Omron CX-Programmer project NewProject (CX-Programmer 9.61)

# PLC NewPLC1: CP1L M

## Global symbols (name address type ; comment)
49.00 BOOL  ; Memória para fazer um movimento horizontal P2 em velocidade lenta até box.
C0017 BOOL  ; Reconhece peça On PH9: st_su_traino_bancalino_deposito_pinza_1.
C0018 BOOL  ; Reconhece peça Off PH9: st_su_traino_bancalino_deposito_pinza_1.
C0350 BOOL  ; Contagem planos mesa de rolos Pinça 2.
H0.06 BOOL  ; Bloqueio descida da ventosa sobre pilha na rulliera (Para formato 120 x 120).
H15.00 BOOL  ; Habilitação formato 120x120 Pinça 1.
T0017 BOOL  ; Reconhece peça On PH9: st_su_traino_bancalino_deposito_pinza_1.
T0018 BOOL  ; Reconhece peça Off PH9: st_su_traino_bancalino_deposito_pinza_1.
T0019 BOOL  ; Tempo desabilita HR0.06 (Habilitação formato 120 x 120).
T0682 BOOL  ; Auxiliar em função da retirada da ftc. PH3: st_pinza_1_ftc_fermata_polmone_3.
T0683 BOOL  ; Auxiliar sobe lento centro.
W0.11 BOOL  ; Reconhece peça sob PH9: st_su_traino_bancalino_deposito_pinza_1.
BIT_11200 112.00 BOOL  ; U32: pinza 1 discesa.
BIT_11201 112.01 BOOL  ; U32: pinza 1 veloce sollevamento.
BIT_11202 112.02 BOOL  ; U41: pinza 2 traslazione_lato_dx / KM9: disponibile.
BIT_11203 112.03 BOOL  ; U41: pinza 2 traslazione_lato_sx / KATB: bareira segurança.
BIT_11204 112.04 BOOL  ; U42: pinza 2 salita.
BIT_11205 112.05 BOOL  ; U42: pinza 2 discesa.
BIT_11207 112.07 BOOL  ; KM32F: pinza 1 freno sollevamento.
BIT_4500 45.00 BOOL  ; Memória Entrada Habilitada Ret Lento SX
BIT_4600 46.00 BOOL  ; Memória Entrada Habilitada Ret Lento DX
BIT_4700 47.00 BOOL  ; Lento Ventosa 1
BIT_4800 48.00 BOOL  ; Exclusão por falta peça SX
BIT_4801 48.01 BOOL  ; Exclusão por falta peça DX
BIT_900 9.00 BOOL  ; SA1: st_ripristino
BIT_901 9.01 BOOL  ; SA2: st_selettore_manuale
BIT_902 9.02 BOOL  ; PM: st_pulsante_marcia
BIT_903 9.03 BOOL  ; PA: st_pulsante_arresto
BIT_904 9.04 BOOL  ; PRA: st_pulsante_reset
BIT_905 9.05 BOOL  ; PX20: st_pinza_1_finecorsa_lato_carico
BIT_906 9.06 BOOL  ; PX21: st_pinza_1_finecorsa_lato_scaric
BIT_907 9.07 BOOL  ; PX22: st_pinza_1_finecorsa_alto
BIT_908 9.08 BOOL  ; PX2: st_pinza_1_finecorsa_basso
BIT_909 9.09 BOOL  ; PH100: st_pinza_1_ftc_per_troppo_pieno_trasporti_uscita
BIT_910 9.10 BOOL  ; PB: st_pinza_1_pulsante_comando_ribaltino
BIT_911 9.11 BOOL  ; CS_Valle: st_consenso_da_valle
CH_A270_Canal_A A270 CHANNEL  ; quota_asse_verticale_pinza2
CH_A271_Canal_B A271 CHANNEL  ; quota_asse_verticale_pinza2
CH_A272_Canal_A A272 CHANNEL  ; quota_asse_verticale_pinza1
CH_A273_Canal_B A273 CHANNEL  ; quota_asse_verticale_pinza1
CNT_100 C0100 BOOL  ; ritardo_fermata_pila_pinza1
CNT_102 C0102 BOOL  ; ritardo_per_deposito_dopo_lettura_ftc_pinza1
CNT_112 C0112 BOOL  ; conteggio_per_deposito_dopo_lettura_ftc_pinza2
CNT_20 C0020 BOOL  ; conteggio_per_stacco_pile
CNT_200 C0200 BOOL  ; intasamento_trasporto_uscita
DM_0 D0 CHANNEL  ; memoria_abilitazione_pinza1
DM_1 D1 CHANNEL  ; memoria_abilitazione_pinza2
DM_10 D10 CHANNEL  ; quota_asse_verticale_pinza1
DM_100 D100 CHANNEL  ; quota_hmi_orizzontale_prelievo_pinza1
DM_102 D102 CHANNEL  ; quota_hmi_verticale_rulliera_prelievo_pinza1
DM_104 D104 CHANNEL  ; quota_hmi_orizzontale_cinghie_deposito_pinza1
DM_106 D106 CHANNEL  ; quota_hmi_verticale_cinghie _deposito_pinza1
DM_108 D108 CHANNEL  ; quot_orizzontale_prelievo_pinza1
DM_110 D110 CHANNEL  ; quota_verticale_rulliera_prelievo_pinza1
DM_112 D112 CHANNEL  ; quota_orizzontale_cinghie_deposito_pinza1
DM_114 D114 CHANNEL  ; quota_verticale_cinghie _deposito_pinza1
DM_116 D116 CHANNEL  ; offset_per_asse_orizzontale_pinza1
DM_118 D118 CHANNEL  ; offset_per_asse_verticale_pinza1
DM_12 D12 CHANNEL  ; quota_asse_orizzontale_pinza1
DM_14 D14 CHANNEL  ; quota_asse_verticale_pinza2
DM_150 D150 CHANNEL  ; tempo_aspiraz_in_prelievo_pinza1
DM_151 D151 CHANNEL  ; Tempo desc Vent 1 M10
DM_152 D152 CHANNEL  ; ritardo_fermata_pila_pinza1
DM_153 D153 CHANNEL  ; ritardo_per_deposito_dopo_lettura_ftc_pinza1
DM_154 D154 CHANNEL  ; conteggio_per_stacco_pile
DM_155 D155 CHANNEL  ; intasamento_trasporto_uscita
DM_16 D16 CHANNEL  ; quota_asse_orizzontale_pinza2
DM_160 D160 CHANNEL  ; tempo_aspiraz_in_prelievo_pinza2
DM_161 D161 CHANNEL  ; tempo_soffio_in_deposito_pinza2
DM_163 D163 CHANNEL  ; ritardo_deposito_su_attesa_pinza2
DM_165 D165 CHANNEL  ; Retardo Lento M10.
DM_2 D2 CHANNEL  ; formato_polmoni
DM_20 D20 CHANNEL  ; offset-_vert_posiz_attesa_su_prelievo_pinza1
DM_200 D200 CHANNEL  ; quota_hmi_orizzontale_prelievo_sx_pinza2
DM_202 D202 CHANNEL  ; quota_hmi_orizzontale_prelievo_dx_pinza2
DM_204 D204 CHANNEL  ; quota_hmi_orizzontale_deposito_pinza2
DM_206 D206 CHANNEL  ; quota_hmi_verticale _deposito_pinza2
DM_208 D208 CHANNEL  ; quota_hmi_verticale_fine_pallet_sx_pinza2
DM_210 D210 CHANNEL  ; quota_hmi_verticale_fine_pallet_dx_pinza2
DM_212 D212 CHANNEL  ; quota_hmi_verticale_pila_completa_pinza2
DM_214 D214 CHANNEL  ; memoria_ultimo_prelievo_pinza2
DM_216 D216 CHANNEL  ; quota_verticale_salita_dopo_prelievo_pinza2
DM_218 D218 CHANNEL  ; quota_verticale_salita_dopo_deposito_pinza2
DM_22 D22 CHANNEL  ; offset+_vert_posiz_attesa_su_prelievo_pinza1
DM_220 D220 CHANNEL  ; quota_orizzontale_prelievo_sx_pinza2
DM_222 D222 CHANNEL  ; quota_orizzontale_prelievo_dx_pinza2
DM_224 D224 CHANNEL  ; quota_orizzontale_deposito_pinza2
DM_226 D226 CHANNEL  ; quota_verticale _deposito_pinza2
DM_228 D228 CHANNEL  ; quota_verticale_fine_pallet_sx_pinza2
DM_230 D230 CHANNEL  ; quota_verticale_fine_pallet_dx_pinza2
DM_232 D232 CHANNEL  ; quota_verticale_pila_completa_pinza2
DM_234 D234 CHANNEL  ; offset_per_asse_orizzontale_pinza2
DM_236 D236 CHANNEL  ; offset_per_asse_verticale_pinza2
DM_24 D24 CHANNEL  ; offset-_orizz_posiz_attesa_su_prelievo_pinza1
DM_250 D250 CHANNEL  ; offset-_orizz_posiz_attesa_su_deposito_pinza2
DM_252 D252 CHANNEL  ; offset+_orizz_posiz_attesa_su_deposito_pinza2
DM_254 D254 CHANNEL  ; offset-_vert_posiz_attesa_su_deposito_pinza2
DM_256 D256 CHANNEL  ; offset+_vert_posiz_attesa_su_deposito_pinza2
DM_258 D258 CHANNEL  ; offset-_orizz_posiz_prelievo_sx_pinza2
DM_26 D26 CHANNEL  ; offset+_orizz_posiz_attesa_su_prelievo_pinza1
DM_260 D260 CHANNEL  ; offset+_orizz_posiz_prelievo_sx_pinza2
DM_262 D262 CHANNEL  ; offset-_orizz_posiz_prelievo_dx_pinza2
DM_264 D264 CHANNEL  ; offset+_orizz_posiz_prelievo_dx_pinza2
DM_266 D266 CHANNEL  ; offset-_vert_posiz_prelievo_pinza2
DM_268 D268 CHANNEL  ; offset+_vert_posiz_prelievo_pinza2
DM_270 D270 CHANNEL  ; offset-_vert_posiz_salita_dopo_prelievo_pinza2
DM_272 D272 CHANNEL  ; offset+_vert_posiz_salita_dopo_prelievo_pinza2
DM_274 D274 CHANNEL  ; offset-_orizz_posiz_deposito_pinza2
DM_276 D276 CHANNEL  ; offset+_orizz_posiz_deposito_pinza2
DM_278 D278 CHANNEL  ; offset-_vert_posiz_attesa_su_deposito_pinza2
DM_28 D28 CHANNEL  ; offset-_orizz_posiz_prelievo_pinza1
DM_280 D280 CHANNEL  ; offset+_vert_posiz_attesa_su_deposito_pinza2
DM_282 D282 CHANNEL  ; offset-_vert_posiz_deposito_pinza2
DM_284 D284 CHANNEL  ; offset+_vert_posiz_deposito_pinza2
DM_286 D286 CHANNEL  ; offset-_vert_posiz_salita_dopo_deposito_pinza2
DM_288 D288 CHANNEL  ; offset+_vert_posiz_salita_dopo_deposito_pinza2
DM_290 D290 CHANNEL  ; step_salita_pinza2
DM_30 D30 CHANNEL  ; offset+_orizz_posiz_prelievo_pinza1
DM_32 D32 CHANNEL  ; offset-_vert_posiz_prelievo_pinza1
DM_34 D34 CHANNEL  ; offset+_vert_posiz_prelievo_pinza1
DM_36 D36 CHANNEL  ; offset-_vert_posiz_salita_dopo_prelievo_pinza1
DM_38 D38 CHANNEL  ; offset
DM_40 D40 CHANNEL  ; offset-_orizz_posiz_deposito_pinza1
DM_400 D400 CHANNEL  ; hz_sollevamento_pinza1_hmi
DM_401 D401 CHANNEL  ; hz_traslazione_pinza1_hmi
DM_402 D402 CHANNEL  ; hz_sollevamento_pinza2_hmi
DM_403 D403 CHANNEL  ; hz_traslazione_pinza2_hmi
DM_42 D42 CHANNEL  ; offset+_orizz_posiz_deposito_pinza1
DM_44 D44 CHANNEL  ; offset-_vert_posiz_attesa_su_deposito_pinza1
DM_450 D450 CHANNEL  ; hz_sollevamento_pinza1_fb
DM_451 D451 CHANNEL  ; hz_traslazione_pinza1_fb
DM_452 D452 CHANNEL  ; hz_sollevamento_pinza2_fb
DM_453 D453 CHANNEL  ; hz_traslazione_pinza2_fb
DM_46 D46 CHANNEL  ; offset+_vert_posiz_attesa_su_deposito_pinza1
DM_48 D48 CHANNEL  ; offset-_vert_posiz_deposito_pinza1
DM_50 D50 CHANNEL  ; offset+_vert_posiz_deposito_pinza1
DM_52 D52 CHANNEL  ; offset-_vert_posiz_salita_dopo_deposito_pinza1
DM_54 D54 CHANNEL  ; offset+_vert_posiz_salita_dopo_deposito_pinza1
DM_56 D56 CHANNEL  ; memoria_ultimo_prelievo_pinza1
DM_58 D58 CHANNEL  ; quota_verticale_salita_dopo_prelievo_pinza1
DM_60 D60 CHANNEL  ; quota_verticale_salita_dopo_deposito_pinza1
DM_62 D62 CHANNEL  ; step_salita_pinza1
HR_0 H0.00 BOOL  ; all_scatto_termico
HR_1 H0.01 BOOL  ; all_inverter
HR_10 H0.10 BOOL  ; Allarme schiacciamento pinza 2.
HR_100 H1.00 BOOL  ; azzerare_assi_pinza2
HR_1000 H10.00 BOOL  ; memoria_conteggio_avvenuto
HR_105 H1.05 BOOL  ; all_pallet_sx_finito
HR_106 H1.06 BOOL  ; all_pallet_dx_finito
HR_107 H1.07 BOOL  ; all_mancanza_pallet
HR_108 H1.08 BOOL  ; all_intrusione_area_sx
HR_109 H1.09 BOOL  ; all_intrusione_area_dx
HR_11 H0.11 BOOL  ; all_intasamento_trasporto_uscita
HR_110 H1.10 BOOL  ; all_micro_sicurezza.
HR_111 H1.11 BOOL  ; all_micro_tasteggio pinza 2.
HR_2 H0.02 BOOL  ; all_aria_compressa
HR_212 H2.12 BOOL  ; Trida_Controle lento nas 3 posições_Sempre On_020323.
HR_213 H2.13 BOOL  ; Trida_Sempre Off_010323.
HR_214 H2.14 BOOL  ; Trida_Sempre Off_050522.
HR_215 H2.15 BOOL  ; Trida_Altura ventosa_210519 (Sempre On).
HR_3 H0.03 BOOL  ; all_consenso_da_valle
HR_4 H0.04 BOOL  ; all_emergenza
HR_5 H0.05 BOOL  ; azzerare_assi_pinza1
HR_50103 H501.03 BOOL  ; polmone_completo
HR_50104 H501.04 BOOL  ; spostamento_quadrotta_da_polmone_a_prelievo
HR_50105 H501.05 BOOL  ; filtro_su_ftc_per_reset_traslazione_quadrotta
HR_8 H0.08 BOOL  ; Allarme micro tasteggio pinza 2.
HR_9 H0.09 BOOL  ; Allarme sicurezza traslazione pinza 2.
IN_0 0.00 BOOL  ; BQ1: Canale A (CH-A270) encoder sollevamento pinza 1.
IN_1 0.01 BOOL  ; BQ1: Canale B (CH-A270) encoder sollevamento pinza 1.
IN_10 0.10 BOOL  ; KABDX: st_pinza_2_barriera_dx_ripristinata (Centralina KABDX - Ok!).
IN_100 1.00 BOOL  ; SQDX: st_pinza_2_sensore_muting_dx (Fc. On durante deslocamento P2 para direita).
IN_101 1.01 BOOL  ; Allarme inverter.
IN_102 1.02 BOOL  ; $?St$Bk?_#[4] / PX102: Ft. Sobreposta Polmone 7 (Ftc. "aérea").$?St$Bk?_#[4]
IN_103 1.03 BOOL  ; Ch. habilitação formato 120 x 120.
IN_104 1.04 BOOL  ; PX104: Intasamento M11 (KM11: traino bancalino deposito pinza 1.) (Parece desativada).
IN_105 1.05 BOOL  ; CH106: parada parcial P1.
IN_106 1.06 BOOL  ; CH106: parada parcial P2.
IN_107 1.07 BOOL  ; Disponibili.
IN_108 1.08 BOOL  ; PE: Bt. emergência.
IN_109 1.09 BOOL  ; Disponibili.
IN_11 0.11 BOOL  ; SQSX: st_pinza_2_sensore_muting_sx (Fc. On durante deslocamento P2 para esquerda).
IN_110 1.10 BOOL  ; SQ100: st_pinza_1_tasteggio_1_presenza_piastrella
IN_111 1.11 BOOL  ; SQ101: st_pinza_1_tasteggio_2_finecorsa.
IN_2 0.02 BOOL  ; BQ2: Canale A (CHA-272) encoder sollevamento pinza 2.
IN_200 2.00 BOOL  ; Disponibili.
IN_201 2.01 BOOL  ; PH1: st_pinza_1_ftc_fermata_polmone_1: bancal operatore (Ribaltatore) (Não tem).
IN_202 2.02 BOOL  ; PH2: st_pinza_1_ftc_fermata_polmone_2.
IN_203 2.03 BOOL  ; PH3: st_pinza_1_ftc_fermata_polmone_3 (Não tem).
IN_204 2.04 BOOL  ; PH4: st_pinza_1_ftc_fermata_polmone_4.
IN_205 2.05 BOOL  ; PH5: st_pinza_1_ftc_fermata_polmone_5.
IN_206 2.06 BOOL  ; PH6: st_pinza_1_ftc_fermata_polmone_6 (Não tem).
IN_207 2.07 BOOL  ; PH7: st_pinza_1_ftc_fermata_polmone_7_lettura_lunghezza_pila (Não tem).
IN_208 2.08 BOOL  ; PH8: st_pinza_1_ftc_fermata_polmone_8_prelievo_pinza_1.
IN_209 2.09 BOOL  ; PH9: st_su_traino_bancalino_deposito_pinza_1.
IN_210 2.10 BOOL  ; PX30: st_reed_ribaltino_alto.
IN_211 2.11 BOOL  ; PX31: st_reed_ribaltino_basso.
IN_3 0.03 BOOL  ; BQ2: Canale B (CHA-272) encoder sollevamento pinza 2.
IN_300 3.00 BOOL  ; P1/P2: st_pressostati.
IN_301 3.01 BOOL  ; PX32: st_pinza_2_finecorsa_lato_pedana_sx.
IN_302 3.02 BOOL  ; PX33: st_pinza_2_finecorsa_lato_pedana_dx.
IN_303 3.03 BOOL  ; PX34: st_pinza_2_finecorsa_alto.
IN_304 3.04 BOOL  ; PX35: st_pinza_2_finecorsa_basso.
IN_305 3.05 BOOL  ; PX36: st_pinza_2_tasteggio_1_presenza_piastrella.
IN_306 3.06 BOOL  ; PH10: st_pinza_2_ftc_presenza_pallet_sx (Sempre On).
IN_307 3.07 BOOL  ; PH11: st_pinza_2_ftc_presenza_pallet_dx (Sempre On).
IN_308 3.08 BOOL  ; P8: st_pinza_2_pulsante_richiesta_accesso_Pedana_sx.
IN_309 3.09 BOOL  ; P9: st_pinza_2_pulsante_richiesta_accesso_pedana_dx.
IN_310 3.10 BOOL  ; Px37: st_pinza_2_tasteggio_2_finecorsa.
IN_311 3.11 BOOL  ; Disponibili.
IN_4 0.04 BOOL  ; BQ3: Canale A (DM14) encoder traslazione pinza 1.
IN_400 4.00 BOOL  ; SA3: st_pinza 2_selettore_esclusione pallet sx.
IN_401 4.01 BOOL  ; SA4: st_pinza 2_selettore_esclusione pallet dx.
IN_402 4.02 BOOL  ; PF: st_pinza 2_pulsante_pila finita.
IN_403 4.03 BOOL  ; PX13: st_pinza_2_presenza_piastrelle.
IN_404 4.04 BOOL  ; Disponibili.
IN_405 4.05 BOOL  ; Disponibili.
IN_406 4.06 BOOL  ; Disponibili.
IN_407 4.07 BOOL  ; Disponibili.
IN_408 4.08 BOOL  ; Disponibili.
IN_409 4.09 BOOL  ; Disponibili.
IN_410 4.10 BOOL  ; Disponibili.
IN_411 4.11 BOOL  ; Disponibili.
IN_5 0.05 BOOL  ; BQ3: Canale B (DM14) encoder traslazione pinza 1.
IN_500 5.00 BOOL  ; SA1: st_ripristino (Sempre On_Jump +).
IN_501 5.01 BOOL  ; SA2: selettore manuale/automatico.
IN_502 5.02 BOOL  ; PM: st_pulsante_marcia.
IN_503 5.03 BOOL  ; PA: st_pulsante_arresto.
IN_504 5.04 BOOL  ; PRA: st_pulsante_reset_allarmi.
IN_505 5.05 BOOL  ; PX20: st_pinza_1_finecorsa_lato_carico.
IN_506 5.06 BOOL  ; PX21: st_pinza_1_finecorsa_lato_scarico.
IN_507 5.07 BOOL  ; PX22: st_pinza_1_finecorsa_alto.
IN_508 5.08 BOOL  ; PX23: st_pinza_1_finecorsa_basso.
IN_509 5.09 BOOL  ; PH100: st_pinza_1_ftc_per_troppo_pieno_trasporti_uscita (Sempre Off_Nada ligado nesta entrada).
IN_510 5.10 BOOL  ; PB: st_pinza_1_pulsante_comando_ribaltino.
IN_511 5.11 BOOL  ; CS_Valle: st_consenso_da_valle.
IN_6 0.06 BOOL  ; BQ4: Canale A (DM16) encoder traslazione pinza 2.
IN_7 0.07 BOOL  ; BQ4: Canale B  (DM16) encoder traslazione pinza 2.
IN_8 0.08 BOOL  ; Allarme termico motori.
IN_9 0.09 BOOL  ; KABSX: St_pinza_2_barriera_sx_ripristinata (Centralina KABSX - Ok!).
OUT_10000 100.00 BOOL  ; KA10: consenso a monte.
OUT_10001 100.01 BOOL  ; HA1: sirena.
OUT_10002 100.02 BOOL  ; HL5: spia allarme.
OUT_10003 100.03 BOOL  ; U32: pinza 1 discesa.
OUT_10004 100.04 BOOL  ; U32: pinza 1 veloce sollevamento.
OUT_10005 100.05 BOOL  ; HL8: spia acesso consentito sx.
OUT_10006 100.06 BOOL  ; HL9: spia acesso consentito dx.
OUT_10007 100.07 BOOL  ; HL10: spia segnalazione pedana sx finita.
OUT_10100 101.00 BOOL  ; HL11: spia segnalazione pedana dx finita.
OUT_10101 101.01 BOOL  ; KM21: pompa vuoto pinza 1.
OUT_10102 101.02 BOOL  ; KA22: pompa vuoto pinza 2.
OUT_10103 101.03 BOOL  ; Clock peças produzidas (Sobre painel Spaccatrice).
OUT_10104 101.04 BOOL  ; U31: pinza 1 traslazione lato scarico.
OUT_10105 101.05 BOOL  ; U31: pinza 1 traslazione lato carico.
OUT_10106 101.06 BOOL  ; U31: pinza 1 veloce traslazione.
OUT_10107 101.07 BOOL  ; U32: pinza1 salita.
OUT_10199 102.00 BOOL  ; Reserva (Desenho elétrico: KM41F: freno traslazione pinza 2).
OUT_10200 102.01 BOOL  ; KM42F: pinza 2 freno solevamento.
OUT_10201 102.02 BOOL  ; KM1: polmone 1: bancalino operatore (Ribaltatore).
OUT_10202 102.03 BOOL  ; KM2: polmone 2.
OUT_10203 102.04 BOOL  ; KM3: polmone 3.
OUT_10204 102.05 BOOL  ; KM4: polmone 4.
OUT_10205 102.06 BOOL  ; KM5: polmone 5.
OUT_10206 102.07 BOOL  ; KM6: polmone 6.
OUT_10300 103.00 BOOL  ; KM7: polmone 7.
OUT_10301 103.01 BOOL  ; KM8: polmone 8 (Sotto pinza 1).
OUT_10302 103.02 BOOL  ; U41: pinza 2 traslazione_lato_dx / KM9: disponibile.
OUT_10303 103.03 BOOL  ; KM10 / KA10403: disponíbile.
OUT_10304 103.04 BOOL  ; KM11: traino bancalino deposito pinza 1.
OUT_10305 103.05 BOOL  ; KM15: disponibile.
OUT_10306 103.06 BOOL  ; U41: pinza 2 traslazione_lato_sx / KATB: barreira segurança.
OUT_10307 103.07 BOOL  ; KASX: acesso pedana sx (On: liberado acesso).
OUT_10400 104.00 BOOL  ; KADX: acesso pedana dx (On: liberado acesso).
OUT_10401 104.01 BOOL  ; KAYV1: ev. salita bancalino operatore.
OUT_10402 104.02 BOOL  ; KAYV2: ev. discesa bancalino operatore.
OUT_10403 104.03 BOOL  ; KAYV3: ev. aspirazione pinza 1.
OUT_10404 104.04 BOOL  ; KAYV4: ev. soffio pinza 1.
OUT_10405 104.05 BOOL  ; KAYV5: ev. aspirazione pinza 2.
OUT_10406 104.06 BOOL  ; KAYV6: ev. soffio pinza 2.
OUT_10407 104.07 BOOL  ; KA10505: disponibile.
OUT_10500 105.00 BOOL  ; Disponibile.
OUT_10501 105.01 BOOL  ; HL12: spia marcia.
OUT_10502 105.02 BOOL  ; U41: pinza 2 veloce traslazione.
OUT_10503 105.03 BOOL  ; U42: pinza 2 veloce solevamento.
OUT_10504 105.04 BOOL  ; U42: pinza 2 salita.
OUT_10505 105.05 BOOL  ; U42: pinza 2 discesa.
OUT_10506 105.06 BOOL  ; Disponibile.
OUT_10507 105.07 BOOL  ; KM32F: pinza 1 freno sollevamento.
TIM_100 T0100 BOOL  ; tempo_aspiraz_in_prelievo_pinza1
TIM_101 T0101 BOOL  ; tempo_soffio_in_deposito_pinza1 Antigo D151
TIM_103 T0103 BOOL  ; attesa_per_rideposito_pinza1
TIM_110 T0110 BOOL  ; tempo_aspiraz_in_prelievo_pinza2
TIM_111 T0111 BOOL  ; tempo_soffio_in_deposito_pinza2
TIM_123 T0123 BOOL  ; attesa_per_rideposito_pinza2
TIM_15 T0015 BOOL  ; Retardo conta peça produzida.
TIM_16 T0016 BOOL  ; Tempo permanência pulso clock.
TIM_20 T0020 BOOL  ; standby_aspiratore_pinza1
TIM_21 T0021 BOOL  ; standby_aspiratpore_pinza2
TIM_25 T0025 BOOL  ; Ret Stop tração de saida
TIM_26 T0026 BOOL  ; Ret FTC Px102 Separa Fila
TIM_27 T0027 BOOL  ; Retardo Lento M10.
TIM_29 T0029 BOOL  ; Tempo Para desligar Bombas com Emergencia
TIM_3 T0003 BOOL  ; Ritardo off st_pinza_1_ftc_fermata_polmone_8_prelievo_pinza_1.
TIM_30 T0030 BOOL  ; Retardo Mivimento Palet Dx Painel
TIM_31 T0031 BOOL  ; Retardo conta peça produzida.
TIM_32 T0032 BOOL  ; Ret. Libera Movimento Palet SX
TIM_33 T0033 BOOL  ; Ret Libera Movimento Palet DX
TIM_34 T0034 BOOL  ; Fim Pilha manual
TIM_35 T0035 BOOL  ; Plano vazio Ventosa 2
TIM_36 T0036 BOOL  ; Ret Leitura Hor SX
TIM_37 T0037 BOOL  ; Ret Leitura Hor DX
TIM_38 T0038 BOOL  ; Retardo libera parada parcial P1.
TIM_39 T0039 BOOL  ; Retardo libera parada parcial P2.
TIM_4 T0004 BOOL  ; Ritardo st_consenso_da_valle
TIM_5 T0005 BOOL  ; Ritardo riconosce pila finita manuale.
TIM_6 T0006 BOOL  ; Ritardo uscita di automatico.
TIM_650 T0650 BOOL  ; ritardo_rich_acc_sx
TIM_651 T0651 BOOL  ; ritardo_rich_acc_dx
TIM_652 T0652 BOOL  ; Ret Libera Acesso DX
TIM_653 T0653 BOOL  ; Ret Libera Acesso SX
TIM_7 T0007 BOOL  ; Ritardo riconosce ftc fermata polmone 6_7.
TIM_8 T0008 BOOL  ; Allarme micro tasteggio pinza 2.
W_0 W0.00 BOOL  ; st_ripristino
W_1 W0.01 BOOL  ; st_scatto_termico
W_10 W0.10 BOOL  ; st_consenso_da_valle senza tempo
W_100 W1.00 BOOL  ; st_pinza_1_finecorsa_lato_carico
W_1000 W10.00 BOOL  ; spia_marcia
W_10000 W100.00 BOOL  ; attesa_per_accesso_sx
W_10002 W100.02 BOOL  ; posizionamento_al_centro_da_rich_acc_sx_dx
W_10003 W100.03 BOOL  ; attesa_sx_con_pinza_a_dx
W_10004 W100.04 BOOL  ; accesso_consentito_a_sx
W_10006 W100.06 BOOL  ; attesa_sx_con_pinza_a_sx
W_1001 W10.01 BOOL  ; spia_allarme
W_10013 W100.13 BOOL  ; allarme_fermo_ciclo
W_10014 W100.14 BOOL  ; tacita_sirena
W_1002 W10.02 BOOL  ; sirena
W_1003 W10.03 BOOL  ; consenso_a_monte
W_101 W1.01 BOOL  ; st_pinza_1_finecorsa_lato_scarico
W_10100 W101.00 BOOL  ; attesa_per_accesso_dx
W_10102 W101.02 BOOL  ; ok_accesso
W_10103 W101.03 BOOL  ; attesa_dx_con_pinza_a_sx
W_10104 W101.04 BOOL  ; accesso_consentito_a_dx
W_10106 W101.06 BOOL  ; attesa_dx_con_pinza_a_dx
W_102 W1.02 BOOL  ; st_pinza_1_rallentamento_lato_carico
W_10203 W102.03 BOOL  ; attesa_ripresa_ciclo
W_103 W1.03 BOOL  ; st_pinza_1_rallentamento_lato_scarico
W_104 W1.04 BOOL  ; st_pinza_1_finecorsa_alto
W_105 W1.05 BOOL  ; st_pinza_1_finecorsa_basso
W_106 W1.06 BOOL  ; st_pinza_1_tasteggio_1_presenza_piastrella
W_107 W1.07 BOOL  ; st_pinza_1_tasteggio_2_finecorsa
W_108 W1.08 BOOL  ; st_pinza_1_ftc_fermata_polmone_8_prelievo_pinza_1.
W_109 W1.09 BOOL  ; st_pinza_1_ftc_lettura_lunghezza_pila
W_110 W1.10 BOOL  ; $?St$Bk?_#[5] / PX102: Ft. Sobreposta Polmone 7 (Ftc. "aérea").$?St$Bk?_#[5]
W_1100 W11.00 BOOL  ; pinza_1_traslazione_verso_carico
W_11000 W110.00 BOOL  ; vel_rallentata_sollevamento_pinza1
W_11001 W110.01 BOOL  ; vel_rallentata_traslazione_pinza1
W_11002 W110.02 BOOL  ; finecorsa_lato_prelievo_pinza1
W_11003 W110.03 BOOL  ; finecorsa_lato_deposito_pinza1
W_1101 W11.01 BOOL  ; pinza_1_traslazione_verso_scarico
W_1102 W11.02 BOOL  ; pinza_1_salita
W_1103 W11.03 BOOL  ; pinza_1_discesa
W_1104 W11.04 BOOL  ; pinza_1_ev_aspirazione
W_1105 W11.05 BOOL  ; pinza_1_ev_soffio
W_1106 W11.06 BOOL  ; pinza_1_aspiratore
W_1107 W11.07 BOOL  ; pinza_1_trasporto1_cinghie
W_1108 W11.08 BOOL  ; pinza_1_trasporto2_cinghie
W_1109 W11.09 BOOL  ; pinza_1_trasporto3_cinghie
W_111 W1.11 BOOL  ; PH5: st_pinza_1_ftc_fermata_polmone_5 (Sem função no programa).
W_1110 W11.10 BOOL  ; Polmone 8 (Sotto pinza 1)_manual.
W_1111 W11.11 BOOL  ; Polmone 7_manual.
W_1112 W11.12 BOOL  ; Polmone 6_manual.
W_1113 W11.13 BOOL  ; Polmone 5_manual.
W_1114 W11.14 BOOL  ; Polmone 4_manual.
W_1115 W11.15 BOOL  ; Polmone 3_manual.
W_112 W1.12 BOOL  ; PH4: st_pinza_1_ftc_fermata_polmone_4.
W_113 W1.13 BOOL  ; PH5: st_pinza_1_ftc_fermata_polmone_5.
W_114 W1.14 BOOL  ; PH2: st_pinza_1_ftc_fermata_polmone_2.
W_115 W1.15 BOOL  ; PH1: st_pinza_1_ftc_fermata_polmone_1: bancal operatore (Ribaltatore) (Não tem).
W_1200 W12.00 BOOL  ; Polmone 2_manual.
W_1201 W12.01 BOOL  ; pinza_1_rulliera_8
W_1202 W12.02 BOOL  ; Polmone 1: bancalino operatore (Ribaltatore)_manual.
W_1203 W12.03 BOOL  ; pinza_1_ev_salita_ribaltino
W_1204 W12.04 BOOL  ; pinza_1_ev_discesa_ribaltino
W_1300 W13.00 BOOL  ; pinza_2_traslazione_da_sx_a_dx
W_1301 W13.01 BOOL  ; pinza_2_traslazione_da_dx_a_sx
W_1302 W13.02 BOOL  ; pinza_2_salita
W_1303 W13.03 BOOL  ; pinza_2_discesa
W_1304 W13.04 BOOL  ; pinza_2_ev_aspirazione
W_1305 W13.05 BOOL  ; pinza_2_ev_soffio
W_1306 W13.06 BOOL  ; pinza_2_aspiratore
W_1307 W13.07 BOOL  ; pinza_2_trasporto1_cinghie
W_1308 W13.08 BOOL  ; pinza_2_trasporto2_cinghie
W_1309 W13.09 BOOL  ; pinza_2_trasporto3_cinghie
W_1310 W13.10 BOOL  ; pinza_2_rulliera_1_deposito
W_1311 W13.11 BOOL  ; pinza_2_rulliera_2
W_1312 W13.12 BOOL  ; pinza_2_rulliera_3
W_1313 W13.13 BOOL  ; pinza_2_trasporto_rulli_deviatore
W_1314 W13.14 BOOL  ; pinza_2_trasporto_cinghie_deviatore
W_1315 W13.15 BOOL  ; pinza_2_ev_deviatore
W_1400 W14.00 BOOL  ; pinza_2_spia_pallet_sx_finito
W_1401 W14.01 BOOL  ; pinza_2_spia_pallet_dx_finito
W_1402 W14.02 BOOL  ; pinza_2_bypass_barriera_sx
W_1403 W14.03 BOOL  ; pinza_2_bypass_barriera_dx
W_1404 W14.04 BOOL  ; pinza_2_spia_accesso_consentito_sx
W_1405 W14.05 BOOL  ; pinza_2_spia_accesso_consentito_dx
W_2 W0.02 BOOL  ; st_allarme_inverter
W_200 W2.00 BOOL  ; st_pinza_1_ftc_fermata_polmone_8
W_2000 W20.00 BOOL  ; spia_marcia_automatico
W_20000 W200.00 BOOL  ; tasto_azzera_assi_pinza1
W_2001 W20.01 BOOL  ; spia_allarme_automatico
W_2002 W20.02 BOOL  ; sirena_automatico
W_2003 W20.03 BOOL  ; consenso_a_monte_automatico
W_201 W2.01 BOOL  ; st_pinza_1_ftc_fermata_polmone_9
W_202 W2.02 BOOL  ; st_pinza_1_pulsante_comando_ribaltino
W_203 W2.03 BOOL  ; st_pinza_1_reed_ribaltino_alto
W_204 W2.04 BOOL  ; st_pinza_1_reed_ribaltino_basso
W_205 W2.05 BOOL  ; PH9: st_su_traino_bancalino_deposito_pinza_1.
W_20500 W205.00 BOOL  ; tasto_azzera_assi_pinza2
W_206 W2.06 BOOL  ; st_pinza_1_ftc_per_troppo_pieno_trasporti_uscita
W_207 W2.07 BOOL  ; st_pinza 2_pulsante_pila finita.
W_208 W2.08 BOOL  ; Sensor presença peça pinza 2.
W_2100 W21.00 BOOL  ; pinza_1_traslazione_verso_carico_automatico
W_21000 W210.00 BOOL  ; vel_rallentata_sollevamento_pinza2
W_21001 W210.01 BOOL  ; vel_rallentata_traslazione_pinza2
W_21002 W210.02 BOOL  ; vel_rallentata_traslazione_pinza2.
W_21003 W210.03 BOOL  ; vel_rallentata_traslazione_pinza2.
W_21004 W210.04 BOOL  ; vel_rallentata_traslazione_pinza2.
W_2101 W21.01 BOOL  ; pinza_1_traslazione_verso_scarico_automatico
W_2102 W21.02 BOOL  ; pinza_1_salita_automatico
W_2103 W21.03 BOOL  ; pinza_1_discesa_automatico
W_2104 W21.04 BOOL  ; pinza_1_ev_aspirazione_automatico
W_2105 W21.05 BOOL  ; pinza_1_ev_soffio_automatico
W_2106 W21.06 BOOL  ; pinza_1_aspiratore_automatico
W_2107 W21.07 BOOL  ; pinza_1_trasporto1_cinghie_automatico
W_2108 W21.08 BOOL  ; pinza_1_trasporto2_cinghie_automatico
W_2109 W21.09 BOOL  ; pinza_1_trasporto3_cinghie_automatico
W_2110 W21.10 BOOL  ; Polmone 8 (Sotto pinza 1)_automatico.
W_21109 W211.09 BOOL  ; posiizonam_al_centro_per_accesso_pinza2
W_2111 W21.11 BOOL  ; Polmone 7._automatico
W_21115 W211.15 BOOL  ; controllo_richieste_accesso
W_2112 W21.12 BOOL  ; Polmone 6_automatico.
W_2113 W21.13 BOOL  ; Polmone 5_automatico.
W_2114 W21.14 BOOL  ; Polmone 4_automatico.
W_2115 W21.15 BOOL  ; Polmone 3_automatico.
W_2200 W22.00 BOOL  ; Polmone 2_automatico.
W_2201 W22.01 BOOL  ; pinza_1_rulliera_8_automatico
W_2202 W22.02 BOOL  ; Polmone 1: bancalino operatore (Ribaltatore)_ribaltino_automatico.
W_2203 W22.03 BOOL  ; pinza_1_ev_salita_ribaltino_automatico
W_2204 W22.04 BOOL  ; pinza_1_ev_discesa_ribaltino_automatico
W_2300 W23.00 BOOL  ; pinza_2_traslazione_da_sx_a_dx_automatico
W_2301 W23.01 BOOL  ; pinza_2_traslazione_da_dx_a_sx_automatico
W_2302 W23.02 BOOL  ; pinza_2_salita_automatico
W_2303 W23.03 BOOL  ; pinza_2_discesa_automatico
W_2304 W23.04 BOOL  ; pinza_2_ev_aspirazione_automatico
W_2305 W23.05 BOOL  ; pinza_2_ev_soffio_automatico
W_2306 W23.06 BOOL  ; pinza_2_aspiratore_automatico
W_2307 W23.07 BOOL  ; pinza_2_trasporto1_cinghie_automatico
W_2308 W23.08 BOOL  ; pinza_2_trasporto2_cinghie_automatico
W_2309 W23.09 BOOL  ; pinza_2_trasporto3_cinghie_automatico
W_2310 W23.10 BOOL  ; pinza_2_rulliera_1_deposito_automatico
W_2311 W23.11 BOOL  ; pinza_2_rulliera_2_automatico
W_2312 W23.12 BOOL  ; pinza_2_rulliera_3_automatico
W_2313 W23.13 BOOL  ; pinza_2_trasporto_rulli_deviatore_automatico
W_2314 W23.14 BOOL  ; pinza_2_trasporto_cinghie_deviatore_automatico
W_2315 W23.15 BOOL  ; pinza_2_ev_deviatore_automatico
W_2400 W24.00 BOOL  ; pinza_2_spia_pallet_sx_finito_automatico
W_2401 W24.01 BOOL  ; pinza_2_spia_pallet_dx_finito_automatico
W_2402 W24.02 BOOL  ; pinza_2_bypass_barriera_sx_automatico
W_2403 W24.03 BOOL  ; pinza_2_bypass_barriera_dx_automatico
W_2404 W24.04 BOOL  ; pinza_2_spia_accesso_consentito_sx_automatico
W_2405 W24.05 BOOL  ; pinza_2_spia_accesso_consentito_dx_automatico
W_27500 W275.00 BOOL  ; flag_presenza_pallet_iniziale
W_3 W0.03 BOOL  ; st_selettore_manuale
W_300 W3.00 BOOL  ; st_pinza_2_finecorsa_lato_sx
W_301 W3.01 BOOL  ; st_pinza_2_finecorsa_lato_dx
W_302 W3.02 BOOL  ; st_pinza_2_finecorsa_alto
W_303 W3.03 BOOL  ; st_pinza_2_finecorsa_basso
W_30309 W303.09 BOOL  ; pallet_sx_esaurito
W_30310 W303.10 BOOL  ; pile_finite_su_rulliera
W_30311 W303.11 BOOL  ; pallet_dx_esaurito
W_30312 W303.12 BOOL  ; Ausiliare esclusione pallet sx.
W_30313 W303.13 BOOL  ; Ausiliare esclusione pallet dx.
W_30314 W303.14 BOOL  ; Ausiliare lento prima discesa su box sx.
W_30315 W303.15 BOOL  ; Ausiliare lento prima discesa su box dx.
W_304 W3.04 BOOL  ; st_pinza_2_tasteggio_1_presenza_piastrella
W_305 W3.05 BOOL  ; st_pinza_2_tasteggio_2_finecorsa
W_306 W3.06 BOOL  ; st_pinza_2_ftc_fermata_prelievo
W_307 W3.07 BOOL  ; st_pinza_2_barriera_sx_ripristinata
W_308 W3.08 BOOL  ; st_pinza_2_barriera_dx_ripristinata
W_309 W3.09 BOOL  ; st_pinza_2_sensore_muting_sx
W_310 W3.10 BOOL  ; st_pinza_2_sensore_muting_dx
W_311 W3.11 BOOL  ; st_pinza_2_pulsante_rich_accesso_sx
W_312 W3.12 BOOL  ; st_pinza_2_pulsante_rich_accesso_dx
W_313 W3.13 BOOL  ; Ausiliare esclusione pallet sx. (Era st_pinza_2_ftc_presenza_pallet_sx).
W_314 W3.14 BOOL  ; Ausiliare esclusione pallet dx. (st_pinza_2_ftc_presenza_pallet_dx).
W_315 W3.15 BOOL  ; st_pinza_2_ftc_su_rulliera_deposito
W_35002 W350.02 BOOL  ; attesa_per_carico_a_sx
W_35003 W350.03 BOOL  ; attesa_per_carico_a_dx
W_35500 W355.00 BOOL  ; pallet_a_a_sx_finito
W_35501 W355.01 BOOL  ; pallet_a_dx_finito
W_35502 W355.02 BOOL  ; pile_finite_stop_ciclo
W_35503 W355.03 BOOL  ; Pila finita manuale.
W_39000 W390.00 BOOL  ; ok_carica_a_sx
W_39001 W390.01 BOOL  ; ok_carica_a_dx
W_4 W0.04 BOOL  ; st_selettore_automatico
W_400 W4.00 BOOL  ; st_pinza_2_ftc_ingresso_deviatore
W_4000 W40.00 BOOL  ; pronto_manuale
W_4001 W40.01 BOOL  ; stato_manuale
W_4002 W40.02 BOOL  ; pronto_automatico
W_4003 W40.03 BOOL  ; stato_automatico
W_4004 W40.04 BOOL  ; standby_pinza1
W_4005 W40.05 BOOL  ; standby_pinza2
W_4007 W40.07 BOOL  ; Retardo Sem Ciclo
W_401 W4.01 BOOL  ; st_pinza_2_ftc_deviatore
W_402 W4.02 BOOL  ; st_pinza_2_ftc_uscita_deviatore
W_403 W4.03 BOOL  ; st_pinza 2_selettore_esclusione pallet sx (On: incluso).
W_404 W4.04 BOOL  ; st_pinza 2_selettore_esclusione pallet dx (On: incluso).
W_410 W4.10 BOOL  ; Formato_1800
W_4100 W41.00 BOOL  ; ciclo_azzeramento_assi_pinza1
W_4101 W41.01 BOOL  ; fine_azzeramento_pinza1
W_4102 W41.02 BOOL  ; flag_assi_azzerati_pinza1
W_4103 W41.03 BOOL  ; salita_per_azzeramento_pinza1
W_4104 W41.04 BOOL  ; discesa_per_azzeramento_pinza1
W_4105 W41.05 BOOL  ; uscita_da_finecorsa_alto_azzeram_pinza1
W_4106 W41.06 BOOL  ; reset_salita_per_azzeramento_pinza1
W_4107 W41.07 BOOL  ; reset_discesa_per_azzeram_pinza1
W_4108 W41.08 BOOL  ; ok_per_azzermento_asse_orizz_pinza1
W_4109 W41.09 BOOL  ; traslazione_lato_carico_per_azzeramento_pinza1
W_4110 W41.10 BOOL  ; traslazione_lato_scarico_per_azzeramento_pinza1
W_4111 W41.11 BOOL  ; reset_traslazione_lato_carico_per_azzeramento_pinza1
W_4112 W41.12 BOOL  ; uscita_da_finec_lato_carico_per_azzeramento_pinza1
W_4113 W41.13 BOOL  ; reset_traslazione_lato_scarico_per_azzeramento_pinza1
W_4300 W43.00 BOOL  ; ciclo_azzeramento_assi_pinza2
W_4301 W43.01 BOOL  ; fine_azzeramento_pinza2
W_4302 W43.02 BOOL  ; flag_assi_azzerati_pinza2
W_4303 W43.03 BOOL  ; salita_per_azzeramento_pinza2
W_4304 W43.04 BOOL  ; discesa_per_azzeramento_pinza2
W_4305 W43.05 BOOL  ; uscita_da_finecorsa_alto_azzeram_pinza2
W_4306 W43.06 BOOL  ; reset_salita_per_azzeramento_pinza2
W_4307 W43.07 BOOL  ; reset_discesa_per_azzeram_pinza2
W_4308 W43.08 BOOL  ; ok_per_azzermento_asse_orizz_pinza2
W_4309 W43.09 BOOL  ; traslazione_lato_sx_per_azzeramento_pinza2
W_4310 W43.10 BOOL  ; traslazione_lato_dx_per_azzeramento_pinza2
W_4311 W43.11 BOOL  ; reset_traslazione_lato_carico_per_azzeramento_pinza2
W_4312 W43.12 BOOL  ; uscita_da_finec_lato_carico_per_azzeramento_pinza2
W_4313 W43.13 BOOL  ; reset_traslazione_lato_scarico_per_azzeramento_pinza2
W_45000 W450.00 BOOL  ; pallet_sx_sostituito
W_45001 W450.01 BOOL  ; pallet_sx_cambiato
W_45002 W450.02 BOOL  ; pallet_dx_sostituito
W_45003 W450.03 BOOL  ; pallet_dx_cambiato
W_5 W0.05 BOOL  ; st_pulsante_marcia
W_5000 W50.00 BOOL  ; start_conteggio_fermata_pila_pinza1
W_50000 W500.00 BOOL  ; start
W_50001 W500.01 BOOL  ; wr_n1
W_50002 W500.02 BOOL  ; busy_n1
W_50003 W500.03 BOOL  ; wr_n2
W_50004 W500.04 BOOL  ; busy_n2
W_50005 W500.05 BOOL  ; wr_n3
W_50006 W500.06 BOOL  ; busy_n3
W_50007 W500.07 BOOL  ; wr_n4
W_50008 W500.08 BOOL  ; busy_n4
W_5001 W50.01 BOOL  ; fermata_polmoni_per_centraggio_
W_50011 W500.11 BOOL  ; restart_write
W_5002 W50.02 BOOL  ; polmonatura_singola
W_5003 W50.03 BOOL  ; polmonatura_doppia
W_5004 W50.04 BOOL  ; polmonatura_per_quadrotta
W_505 W5.05 BOOL  ; Espelho st_pinza_2_tasteggio_2_finecorsa
W_6 W0.06 BOOL  ; st_pulsante_arresto
W_6000 W60.00 BOOL  ; abilitazione_pinza1
W_6001 W60.01 BOOL  ; richiesta_inizio_ciclo_pinza1
W_6002 W60.02 BOOL  ; pinza1_in_ciclo
W_6003 W60.03 BOOL  ; start_ciclo_pinza1
W_6008 W60.08 BOOL  ; primo_ciclo_pinza1
W_6100 W61.00 BOOL  ; posizione_attesa_su_prelievo_pinza1
W_6101 W61.01 BOOL  ; posiz_attesa_su_prelievo_discesa_pinza1
W_6102 W61.02 BOOL  ; posiz_attesa_su_prelievo_salita_pinza1
W_6103 W61.03 BOOL  ; ok_posione_verticale_attesa_pinza1
W_6104 W61.04 BOOL  ; posiz_attesa_su_prelievo_trasl_verso_deposito_pinza1
W_6105 W61.05 BOOL  ; posiz_attesa_su_prelievo_trasl_verso_carico_pinza1
W_6106 W61.06 BOOL  ; ok_posione_orizzontale_attesa_pinza1
W_6200 W62.00 BOOL  ; posizione_prelievo_asse_orizzontale_pinza1
W_6201 W62.01 BOOL  ; posiz_prelievo_trasl_verso_deposito_pinza1
W_6202 W62.02 BOOL  ; posiz_prelievo_trasl_verso_prelievo_pinza1
W_6203 W62.03 BOOL  ; ok_posione_orizzontale_prelievo_pinza1
W_6300 W63.00 BOOL  ; discesa_per_prelievo_piastrella_pinza1
W_6301 W63.01 BOOL  ; piastrella_su_ventose_pinza1
W_6302 W63.02 BOOL  ; posizione_verticale_discesa_prelievo_pinza1
W_6303 W63.03 BOOL  ; ok_posizione_verticale_prelievo_pinza1
W_6304 W63.04 BOOL  ; ok_posizione_verticale_rideposito_su_prelievo_pinza1
W_6400 W64.00 BOOL  ; prelievo_piastrella_pinza1
W_6401 W64.01 BOOL  ; aspirazione_per_prelievo_pinza1
W_6402 W64.02 BOOL  ; ok_prelievo_pinza1
W_6500 W65.00 BOOL  ; salita_dopo_prelievo_piastrella_pinza1
W_6501 W65.01 BOOL  ; posizionamento_verticale_salita_dopo_prelievo_pinza1
W_6502 W65.02 BOOL  ; posizionamento_verticale_discesa_dopo_prelievo_pinza1
W_6503 W65.03 BOOL  ; ok_posizione_verticale_dopo_prelievo_pinza1
W_6600 W66.00 BOOL  ; posizione_deposito_asse_orizzontale_pinza1
W_6601 W66.01 BOOL  ; posizionamento_orizzontale_verso_deposito_per_deposito_pinza1
W_6602 W66.02 BOOL  ; posizionamento_orizzontale_verso_prelievo_per_deposito_pinza1
W_6603 W66.03 BOOL  ; ok_posizione_orizzontale_deposito_pinza1
W_6700 W67.00 BOOL  ; discesa_per_attesa_deposito_pinza1
W_6701 W67.01 BOOL  ; posizionamento_verticale_salita_per_attesa_su_deposito_pinza1
W_6702 W67.02 BOOL  ; posizionamento_verticale_discesa_per_attesa_su_deposito_pinza1
W_6703 W67.03 BOOL  ; ok_posizionamento_verticale_attesa_deposito_pinza1
W_6800 W68.00 BOOL  ; discesa_per_deposito_piastrella_pinza1
W_6801 W68.01 BOOL  ; posizionamento_verticale_salita_per_deposito_pinza1
W_6802 W68.02 BOOL  ; posizionamento_verticale_discesa_per_deposito_pinza1
W_6803 W68.03 BOOL  ; ok_posizione_verticale_deposito_pinza1
W_6900 W69.00 BOOL  ; deposito_piastrella_pinza1
W_6901 W69.01 BOOL  ; soffio_per_deposito_pinza1
W_6902 W69.02 BOOL  ; ok_deposito_pinza1
W_7 W0.07 BOOL  ; st_pulsante_reset
W_7000 W70.00 BOOL  ; salita_dopo_deposito_pinza1
W_7001 W70.01 BOOL  ; posizionamento_verticale_salita_dopo_deposito_pinza1
W_7002 W70.02 BOOL  ; posizionamento_verticale_discesa_dopo_deposito_pinza1
W_7003 W70.03 BOOL  ; ok_posizione_veticale_dopo_deposito_pinza1
W_7100 W71.00 BOOL  ; reset_tutti_cicli_pinza1
W_7101 W71.01 BOOL  ; ciclo_di_rideposito_pinza1
W_7102 W71.02 BOOL  ; memoria_ciclo_rideposito
W_8 W0.08 BOOL  ; st_consenso_da_valle con tempo.
W_8000 W80.00 BOOL  ; abilitazione_pinza2
W_8001 W80.01 BOOL  ; richiesta_inizio_ciclo_pinza2
W_8002 W80.02 BOOL  ; pinza2_in_ciclo
W_8003 W80.03 BOOL  ; start_ciclo_pinza2
W_8004 W80.04 BOOL  ; rischiesta_accesso_in_corso_con_fermo_ciclo
W_8005 W80.05 BOOL  ; rischiesta_accesso_in_corso_senza_fermo_ciclo
W_8006 W80.06 BOOL  ; abilita_pallet_sx
W_8007 W80.07 BOOL  ; abilita_pallet_dx
W_8008 W80.08 BOOL  ; primo_ciclo_rallentato_pinza_2
W_8009 W80.09 BOOL  ; primo_ciclo_pinza_2
W_8100 W81.00 BOOL  ; posizione_attesa_su_deposito_pinza2
W_8101 W81.01 BOOL  ; posiz_attesa_su_deposito_discesa_pinza2
W_8102 W81.02 BOOL  ; posiz_attesa_su_deposito_salita_pinza2
W_8103 W81.03 BOOL  ; ok_posione_verticale_attesa_pinza2
W_8104 W81.04 BOOL  ; posiz_attesa_su_deposito_trasl_verso_dx_pinza2
W_8105 W81.05 BOOL  ; posiz_attesa_su_deposito_trasl_verso_sx_pinza2
W_8106 W81.06 BOOL  ; ok_posione_orizzontale_attesa_pinza2
W_8107 W81.07 BOOL  ; deposito_piastrella_da_ciclo_rimasta_su_ventose
W_8200 W82.00 BOOL  ; posizione_prelievo_asse_orizzontale_pinza2
W_8201 W82.01 BOOL  ; posiz_prelievo_sx_trasl_verso_dx_pinza2 (Sempre off).
W_8202 W82.02 BOOL  ; posiz_prelievo_sx_trasl_verso_sx_pinza2
W_8203 W82.03 BOOL  ; ok_posione_orizzontale_prelievo_sx_pinza2
W_8204 W82.04 BOOL  ; posiz_prelievo_dx_trasl_verso_dx_pinza2
W_8205 W82.05 BOOL  ; posiz_prelievo_dx_trasl_verso_sx_pinza2
W_8206 W82.06 BOOL  ; ok_posione_orizzontale_prelievo_dx_pinza2
W_8300 W83.00 BOOL  ; discesa_per_prelievo_piastrella_pinza2
W_8301 W83.01 BOOL  ; piastrella_su_ventose_pinza2
W_8302 W83.02 BOOL  ; posizione_verticale_discesa_prelievo_pinza2
W_8303 W83.03 BOOL  ; ok_posizione_verticale_prelievo_pinza2
W_8304 W83.04 BOOL  ; ok_posizione_verticale_rideposito_su_prelievo_pinza2
W_8400 W84.00 BOOL  ; prelievo_piastrella_pinza2
W_8401 W84.01 BOOL  ; aspirazione_per_prelievo_pinza2
W_8402 W84.02 BOOL  ; ok_prelievo_pinza2
W_8500 W85.00 BOOL  ; salita_dopo_prelievo_piastrella_pinza2
W_8501 W85.01 BOOL  ; posizionamento_verticale_salita_dopo_prelievo_pinza2
W_8502 W85.02 BOOL  ; posizionamento_verticale_discesa_dopo_prelievo_pinza2
W_8503 W85.03 BOOL  ; ok_posizione_verticale_dopo_prelievo_pinza2
W_8600 W86.00 BOOL  ; posizione_deposito_asse_orizzontale_pinza2
W_8601 W86.01 BOOL  ; posizionamento_orizzontale_verso_dx_per_deposito_pinza2
W_8602 W86.02 BOOL  ; posizionamento_orizzontale_verso_sx_per_deposito_pinza2
W_8603 W86.03 BOOL  ; ok_posizione_orizzontale_deposito_pinza2
W_8700 W87.00 BOOL  ; discesa_per_attesa_deposito_pinza2
W_8701 W87.01 BOOL  ; posizionamento_verticale_salita_per_attesa_su_deposito_pinza2
W_8702 W87.02 BOOL  ; posizionamento_verticale_discesa_per_attesa_su_deposito_pinza2
W_8703 W87.03 BOOL  ; ok_posizionamento_verticale_attesa_deposito_pinza2
W_8800 W88.00 BOOL  ; discesa_per_deposito_piastrella_pinza2
W_8801 W88.01 BOOL  ; posizionamento_verticale_salita_per_deposito_pinza2
W_8802 W88.02 BOOL  ; posizionamento_verticale_discesa_per_deposito_pinza2
W_8803 W88.03 BOOL  ; ok_posizione_verticale_deposito_pinza2
W_8900 W89.00 BOOL  ; deposito_piastrella_pinza2
W_8901 W89.01 BOOL  ; soffio_per_deposito_pinza2
W_8902 W89.02 BOOL  ; ok_deposito_pinza2
W_8903 W89.03 BOOL  ; Ausiliare per blocco traslazione pinza 2.
W_9 W0.09 BOOL  ; st_pressostato
W_9000 W90.00 BOOL  ; salita_dopo_deposito_pinza2
W_9001 W90.01 BOOL  ; posizionamento_verticale_salita_dopo_deposito_pinza2
W_9002 W90.02 BOOL  ; posizionamento_verticale_discesa_dopo_deposito_pinza2
W_9003 W90.03 BOOL  ; ok_posizione_veticale_dopo_deposito_pinza2
W_9100 W91.00 BOOL  ; reset_tutti_cicli_pinza2
W_9101 W91.01 BOOL  ; ciclo_di_rideposito_pinza2
wr_n1 Modbus_Write_Parameter
wr_n2 Modbus_Write_Parameter
wr_n3 Modbus_Write_Parameter
wr_n4 Modbus_Write_Parameter

## Program NuovoProgramma1 (cyclic task 0)
Local symbols
DM_308 DINT

### Section task_interrupt

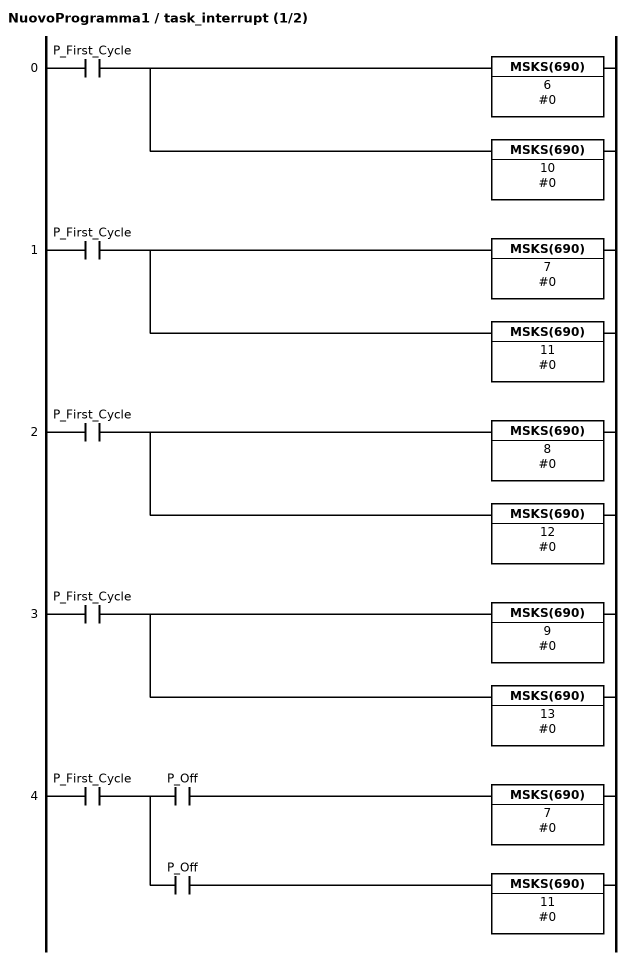
; rung 0
LD P_First_Cycle
MSKS(690) 6 #0
MSKS(690) 10 #0
; rung 1
LD P_First_Cycle
MSKS(690) 7 #0
MSKS(690) 11 #0
; rung 2
LD P_First_Cycle
MSKS(690) 8 #0
MSKS(690) 12 #0
; rung 3
LD P_First_Cycle
MSKS(690) 9 #0
MSKS(690) 13 #0
; rung 4
LD P_First_Cycle
OUT TR0
AND P_Off
MSKS(690) 7 #0
LD TR0
AND P_Off
MSKS(690) 11 #0

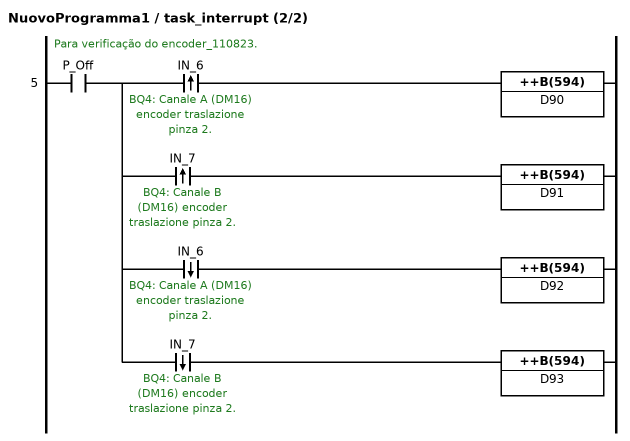
; rung 5: Para verificação do encoder_110823.
LD P_Off
OUT TR0
@AND IN_6  ; BQ4: Canale A (DM16) encoder traslazione pinza 2.
++B(594) D90
LD TR0
@AND IN_7  ; BQ4: Canale B  (DM16) encoder traslazione pinza 2.
++B(594) D91
LD TR0
%AND IN_6  ; BQ4: Canale A (DM16) encoder traslazione pinza 2.
++B(594) D92
LD TR0
%AND IN_7  ; BQ4: Canale B  (DM16) encoder traslazione pinza 2.
++B(594) D93

### Section interfaccia_input

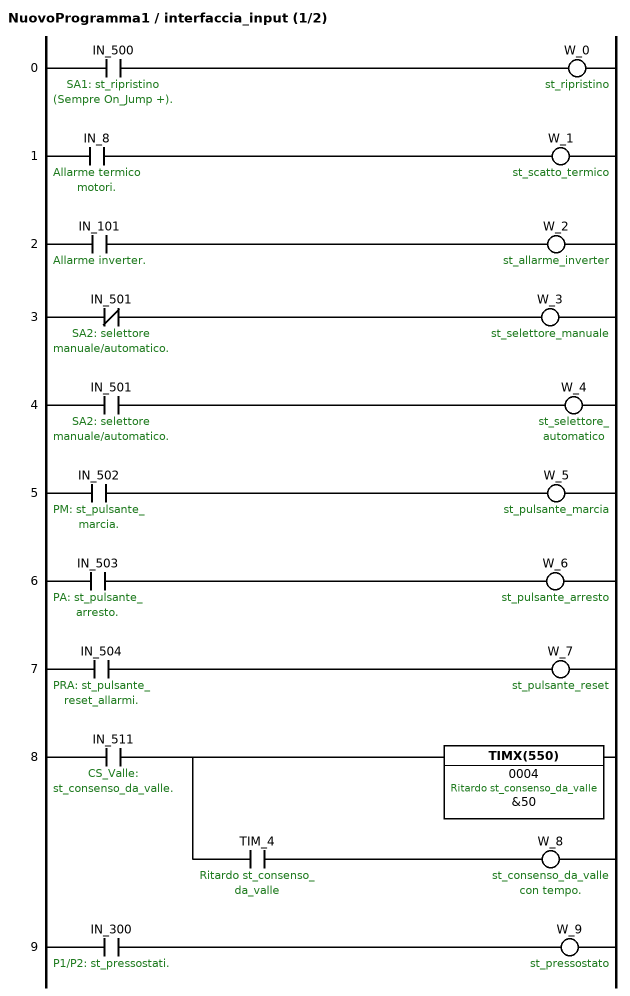
; rung 0
LD IN_500  ; SA1: st_ripristino (Sempre On_Jump +).
OUT W_0  ; st_ripristino
; rung 1
LD IN_8  ; Allarme termico motori.
OUT W_1  ; st_scatto_termico
; rung 2
LD IN_101  ; Allarme inverter.
OUT W_2  ; st_allarme_inverter
; rung 3
LDNOT IN_501  ; SA2: selettore manuale/automatico.
OUT W_3  ; st_selettore_manuale
; rung 4
LD IN_501  ; SA2: selettore manuale/automatico.
OUT W_4  ; st_selettore_automatico
; rung 5
LD IN_502  ; PM: st_pulsante_marcia.
OUT W_5  ; st_pulsante_marcia
; rung 6
LD IN_503  ; PA: st_pulsante_arresto.
OUT W_6  ; st_pulsante_arresto
; rung 7
LD IN_504  ; PRA: st_pulsante_reset_allarmi.
OUT W_7  ; st_pulsante_reset
; rung 8
LD IN_511  ; CS_Valle: st_consenso_da_valle.
TIMX(550) 0004 &50  ; Ritardo st_consenso_da_valle
AND TIM_4  ; Ritardo st_consenso_da_valle
OUT W_8  ; st_consenso_da_valle con tempo.
; rung 9
LD IN_300  ; P1/P2: st_pressostati.
OUT W_9  ; st_pressostato

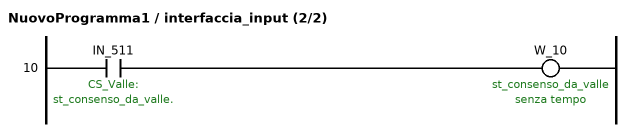
; rung 10
LD IN_511  ; CS_Valle: st_consenso_da_valle.
OUT W_10  ; st_consenso_da_valle senza tempo

### Section interfaccia_input_pinza_ribaltino

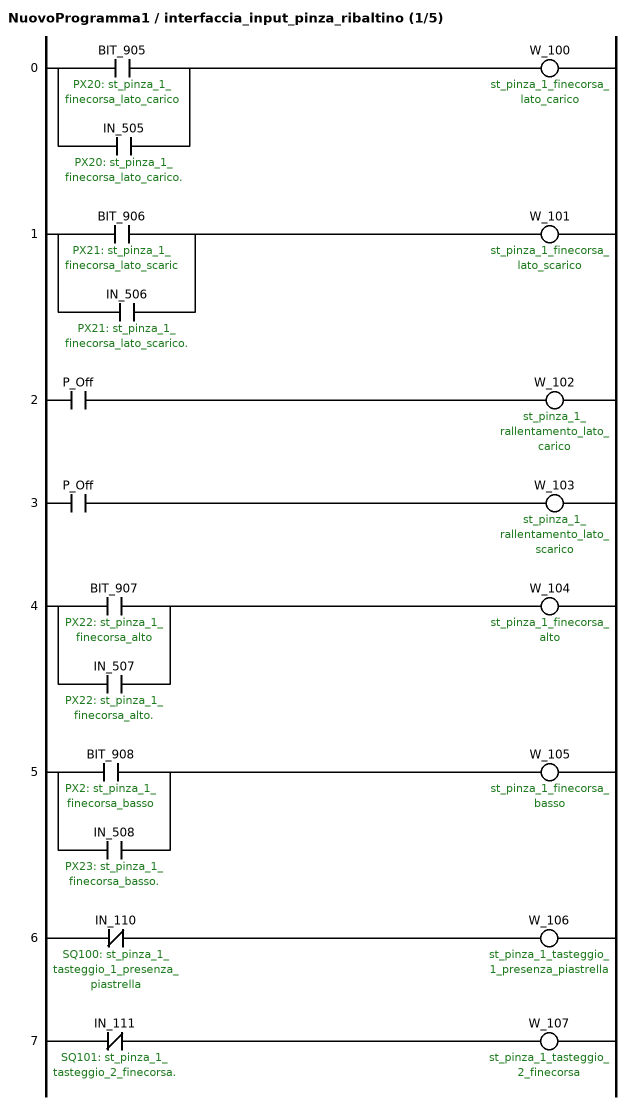
; rung 0
LD BIT_905  ; PX20: st_pinza_1_finecorsa_lato_carico
OR IN_505  ; PX20: st_pinza_1_finecorsa_lato_carico.
OUT W_100  ; st_pinza_1_finecorsa_lato_carico
; rung 1
LD BIT_906  ; PX21: st_pinza_1_finecorsa_lato_scaric
OR IN_506  ; PX21: st_pinza_1_finecorsa_lato_scarico.
OUT W_101  ; st_pinza_1_finecorsa_lato_scarico
; rung 2
LD P_Off
OUT W_102  ; st_pinza_1_rallentamento_lato_carico
; rung 3
LD P_Off
OUT W_103  ; st_pinza_1_rallentamento_lato_scarico
; rung 4
LD BIT_907  ; PX22: st_pinza_1_finecorsa_alto
OR IN_507  ; PX22: st_pinza_1_finecorsa_alto.
OUT W_104  ; st_pinza_1_finecorsa_alto
; rung 5
LD BIT_908  ; PX2: st_pinza_1_finecorsa_basso
OR IN_508  ; PX23: st_pinza_1_finecorsa_basso.
OUT W_105  ; st_pinza_1_finecorsa_basso
; rung 6
LDNOT IN_110  ; SQ100: st_pinza_1_tasteggio_1_presenza_piastrella
OUT W_106  ; st_pinza_1_tasteggio_1_presenza_piastrella
; rung 7
LDNOT IN_111  ; SQ101: st_pinza_1_tasteggio_2_finecorsa.
OUT W_107  ; st_pinza_1_tasteggio_2_finecorsa

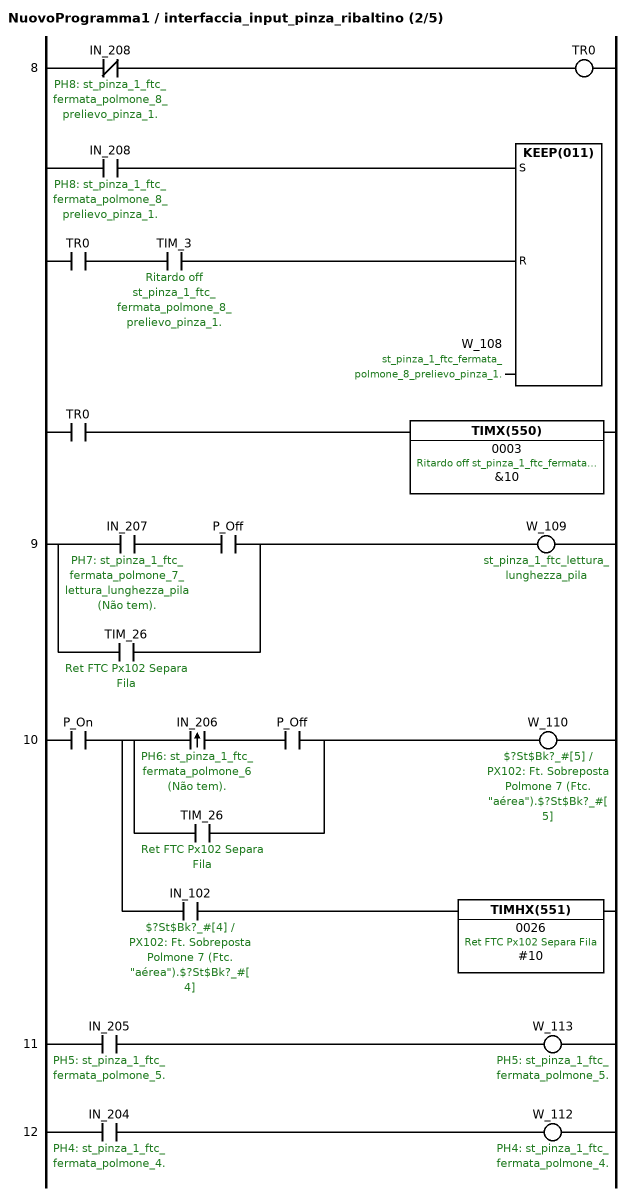
; rung 8
LD IN_208  ; PH8: st_pinza_1_ftc_fermata_polmone_8_prelievo_pinza_1.
LDNOT IN_208  ; PH8: st_pinza_1_ftc_fermata_polmone_8_prelievo_pinza_1.
OUT TR0
AND TIM_3  ; Ritardo off st_pinza_1_ftc_fermata_polmone_8_prelievo_pinza_1.
KEEP(011) W_108  ; st_pinza_1_ftc_fermata_polmone_8_prelievo_pinza_1.
LD TR0
TIMX(550) 0003 &10  ; Ritardo off st_pinza_1_ftc_fermata_polmone_8_prelievo_pinza_1.
; rung 9
LD IN_207  ; PH7: st_pinza_1_ftc_fermata_polmone_7_lettura_lunghezza_pila (Não tem).
AND P_Off
OR TIM_26  ; Ret FTC Px102 Separa Fila
OUT W_109  ; st_pinza_1_ftc_lettura_lunghezza_pila
; rung 10
LD P_On
OUT TR0
@LD IN_206  ; PH6: st_pinza_1_ftc_fermata_polmone_6 (Não tem).
AND P_Off
OR TIM_26  ; Ret FTC Px102 Separa Fila
ANDLD
OUT W_110  ; $?St$Bk?_#[5] / PX102: Ft. Sobreposta Polmone 7 (Ftc. "aérea").$?St$Bk?_#[5]
LD TR0
AND IN_102  ; $?St$Bk?_#[4] / PX102: Ft. Sobreposta Polmone 7 (Ftc. "aérea").$?St$Bk?_#[4]
TIMHX(551) 0026 #10  ; Ret FTC Px102 Separa Fila
; rung 11
LD IN_205  ; PH5: st_pinza_1_ftc_fermata_polmone_5.
OUT W_113  ; PH5: st_pinza_1_ftc_fermata_polmone_5.
; rung 12
LD IN_204  ; PH4: st_pinza_1_ftc_fermata_polmone_4.
OUT W_112  ; PH4: st_pinza_1_ftc_fermata_polmone_4.

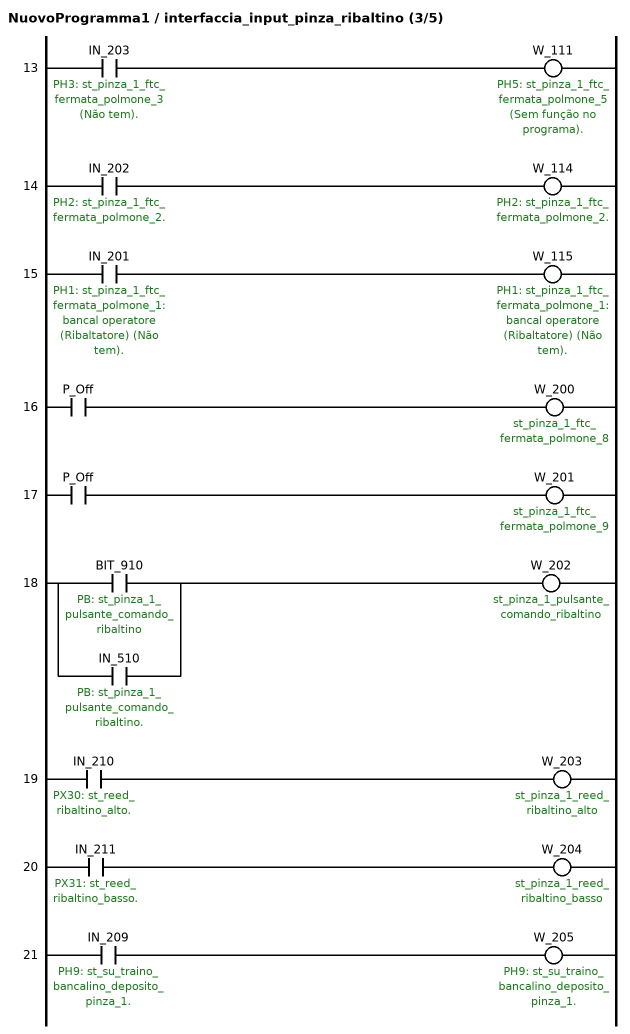
; rung 13
LD IN_203  ; PH3: st_pinza_1_ftc_fermata_polmone_3 (Não tem).
OUT W_111  ; PH5: st_pinza_1_ftc_fermata_polmone_5 (Sem função no programa).
; rung 14
LD IN_202  ; PH2: st_pinza_1_ftc_fermata_polmone_2.
OUT W_114  ; PH2: st_pinza_1_ftc_fermata_polmone_2.
; rung 15
LD IN_201  ; PH1: st_pinza_1_ftc_fermata_polmone_1: bancal operatore (Ribaltatore) (Não tem).
OUT W_115  ; PH1: st_pinza_1_ftc_fermata_polmone_1: bancal operatore (Ribaltatore) (Não tem).
; rung 16
LD P_Off
OUT W_200  ; st_pinza_1_ftc_fermata_polmone_8
; rung 17
LD P_Off
OUT W_201  ; st_pinza_1_ftc_fermata_polmone_9
; rung 18
LD BIT_910  ; PB: st_pinza_1_pulsante_comando_ribaltino
OR IN_510  ; PB: st_pinza_1_pulsante_comando_ribaltino.
OUT W_202  ; st_pinza_1_pulsante_comando_ribaltino
; rung 19
LD IN_210  ; PX30: st_reed_ribaltino_alto.
OUT W_203  ; st_pinza_1_reed_ribaltino_alto
; rung 20
LD IN_211  ; PX31: st_reed_ribaltino_basso.
OUT W_204  ; st_pinza_1_reed_ribaltino_basso
; rung 21
LD IN_209  ; PH9: st_su_traino_bancalino_deposito_pinza_1.
OUT W_205  ; PH9: st_su_traino_bancalino_deposito_pinza_1.

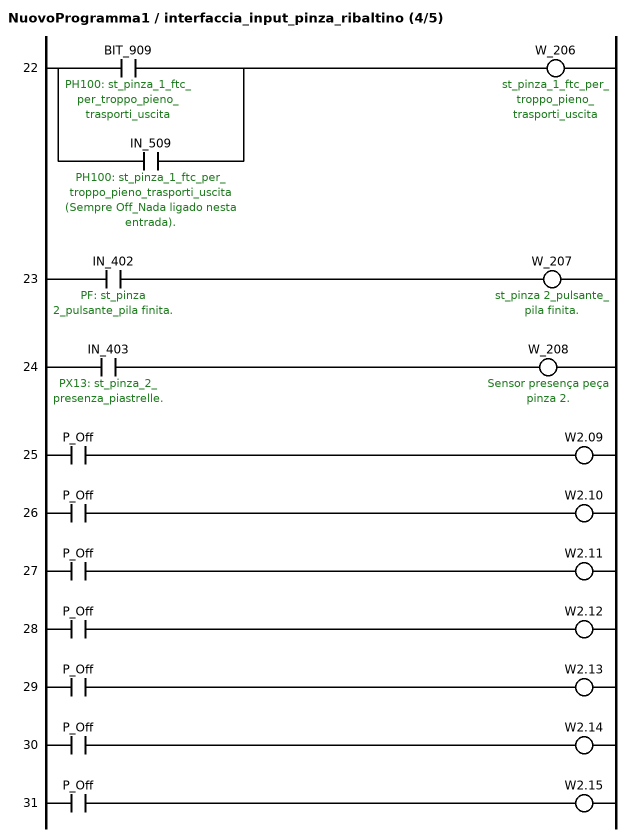
; rung 22
LD BIT_909  ; PH100: st_pinza_1_ftc_per_troppo_pieno_trasporti_uscita
OR IN_509  ; PH100: st_pinza_1_ftc_per_troppo_pieno_trasporti_uscita (Sempre Off_Nada ligado nesta entrada).
OUT W_206  ; st_pinza_1_ftc_per_troppo_pieno_trasporti_uscita
; rung 23
LD IN_402  ; PF: st_pinza 2_pulsante_pila finita.
OUT W_207  ; st_pinza 2_pulsante_pila finita.
; rung 24
LD IN_403  ; PX13: st_pinza_2_presenza_piastrelle.
OUT W_208  ; Sensor presença peça pinza 2.
; rung 25
LD P_Off
OUT W2.09
; rung 26
LD P_Off
OUT W2.10
; rung 27
LD P_Off
OUT W2.11
; rung 28
LD P_Off
OUT W2.12
; rung 29
LD P_Off
OUT W2.13
; rung 30
LD P_Off
OUT W2.14
; rung 31
LD P_Off
OUT W2.15

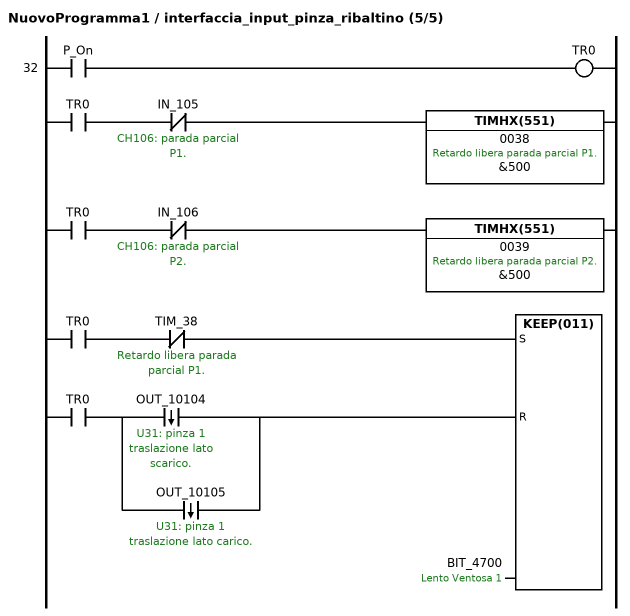
; rung 32
LD P_On
OUT TR0
ANDNOT IN_105  ; CH106: parada parcial P1.
TIMHX(551) 0038 &500  ; Retardo libera parada parcial P1.
LD TR0
ANDNOT IN_106  ; CH106: parada parcial P2.
TIMHX(551) 0039 &500  ; Retardo libera parada parcial P2.
LD TR0
ANDNOT TIM_38  ; Retardo libera parada parcial P1.
LD TR0
%LD OUT_10104  ; U31: pinza 1 traslazione lato scarico.
%OR OUT_10105  ; U31: pinza 1 traslazione lato carico.
ANDLD
KEEP(011) BIT_4700  ; Lento Ventosa 1

### Section interfaccia_input_pinza_pallet

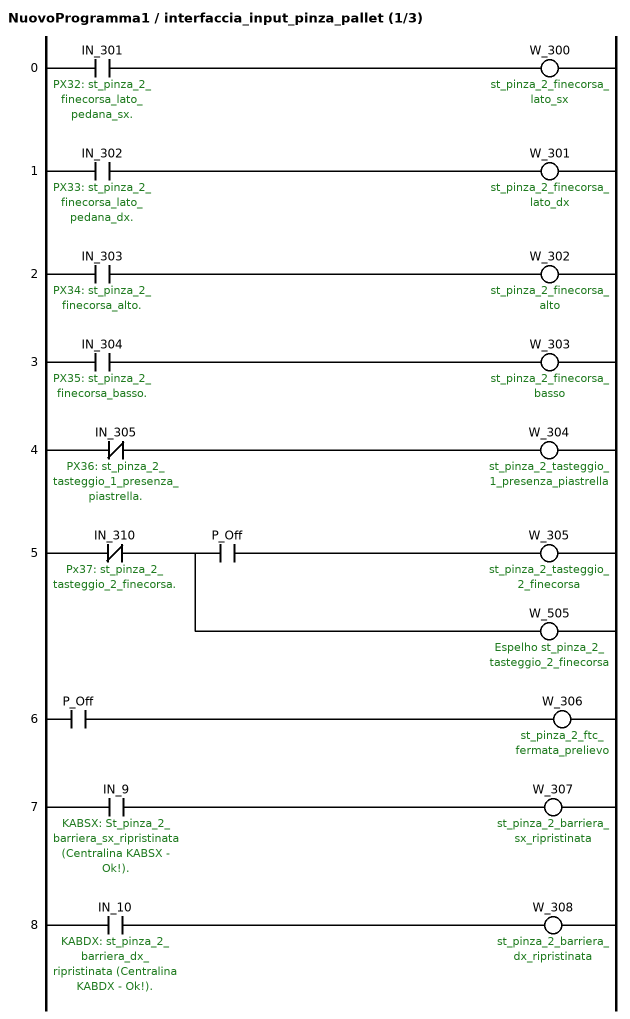
; rung 0
LD IN_301  ; PX32: st_pinza_2_finecorsa_lato_pedana_sx.
OUT W_300  ; st_pinza_2_finecorsa_lato_sx
; rung 1
LD IN_302  ; PX33: st_pinza_2_finecorsa_lato_pedana_dx.
OUT W_301  ; st_pinza_2_finecorsa_lato_dx
; rung 2
LD IN_303  ; PX34: st_pinza_2_finecorsa_alto.
OUT W_302  ; st_pinza_2_finecorsa_alto
; rung 3
LD IN_304  ; PX35: st_pinza_2_finecorsa_basso.
OUT W_303  ; st_pinza_2_finecorsa_basso
; rung 4
LDNOT IN_305  ; PX36: st_pinza_2_tasteggio_1_presenza_piastrella.
OUT W_304  ; st_pinza_2_tasteggio_1_presenza_piastrella
; rung 5
LDNOT IN_310  ; Px37: st_pinza_2_tasteggio_2_finecorsa.
OUT TR0
AND P_Off
OUT W_305  ; st_pinza_2_tasteggio_2_finecorsa
LD TR0
OUT W_505  ; Espelho st_pinza_2_tasteggio_2_finecorsa
; rung 6
LD P_Off
OUT W_306  ; st_pinza_2_ftc_fermata_prelievo
; rung 7
LD IN_9  ; KABSX: St_pinza_2_barriera_sx_ripristinata (Centralina KABSX - Ok!).
OUT W_307  ; st_pinza_2_barriera_sx_ripristinata
; rung 8
LD IN_10  ; KABDX: st_pinza_2_barriera_dx_ripristinata (Centralina KABDX - Ok!).
OUT W_308  ; st_pinza_2_barriera_dx_ripristinata

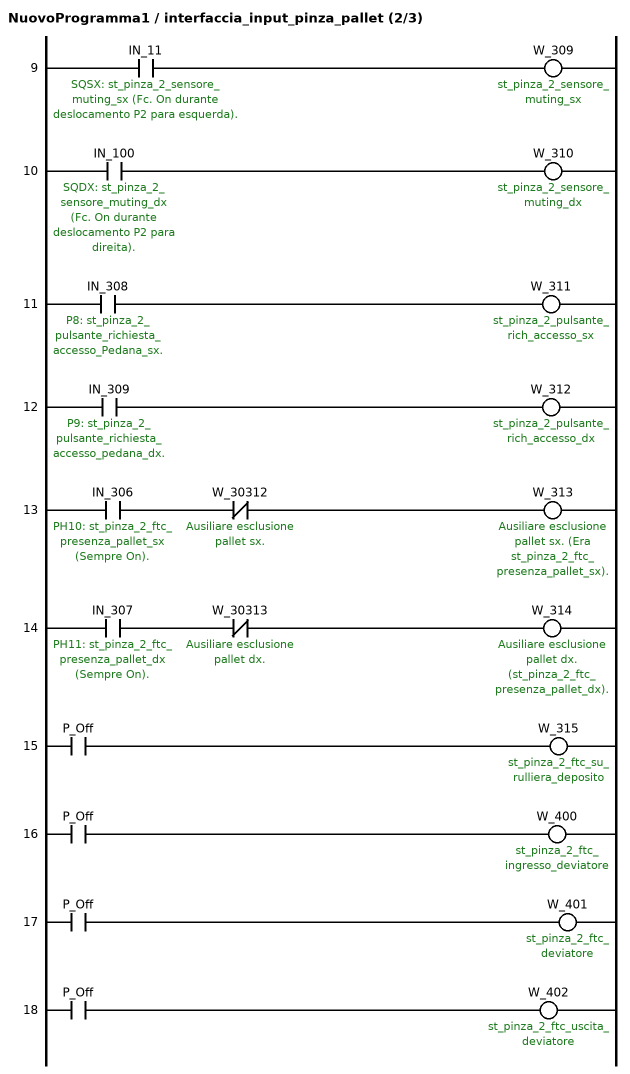
; rung 9
LD IN_11  ; SQSX: st_pinza_2_sensore_muting_sx (Fc. On durante deslocamento P2 para esquerda).
OUT W_309  ; st_pinza_2_sensore_muting_sx
; rung 10
LD IN_100  ; SQDX: st_pinza_2_sensore_muting_dx (Fc. On durante deslocamento P2 para direita).
OUT W_310  ; st_pinza_2_sensore_muting_dx
; rung 11
LD IN_308  ; P8: st_pinza_2_pulsante_richiesta_accesso_Pedana_sx.
OUT W_311  ; st_pinza_2_pulsante_rich_accesso_sx
; rung 12
LD IN_309  ; P9: st_pinza_2_pulsante_richiesta_accesso_pedana_dx.
OUT W_312  ; st_pinza_2_pulsante_rich_accesso_dx
; rung 13
LD IN_306  ; PH10: st_pinza_2_ftc_presenza_pallet_sx (Sempre On).
ANDNOT W_30312  ; Ausiliare esclusione pallet sx.
OUT W_313  ; Ausiliare esclusione pallet sx. (Era st_pinza_2_ftc_presenza_pallet_sx).
; rung 14
LD IN_307  ; PH11: st_pinza_2_ftc_presenza_pallet_dx (Sempre On).
ANDNOT W_30313  ; Ausiliare esclusione pallet dx.
OUT W_314  ; Ausiliare esclusione pallet dx. (st_pinza_2_ftc_presenza_pallet_dx).
; rung 15
LD P_Off
OUT W_315  ; st_pinza_2_ftc_su_rulliera_deposito
; rung 16
LD P_Off
OUT W_400  ; st_pinza_2_ftc_ingresso_deviatore
; rung 17
LD P_Off
OUT W_401  ; st_pinza_2_ftc_deviatore
; rung 18
LD P_Off
OUT W_402  ; st_pinza_2_ftc_uscita_deviatore

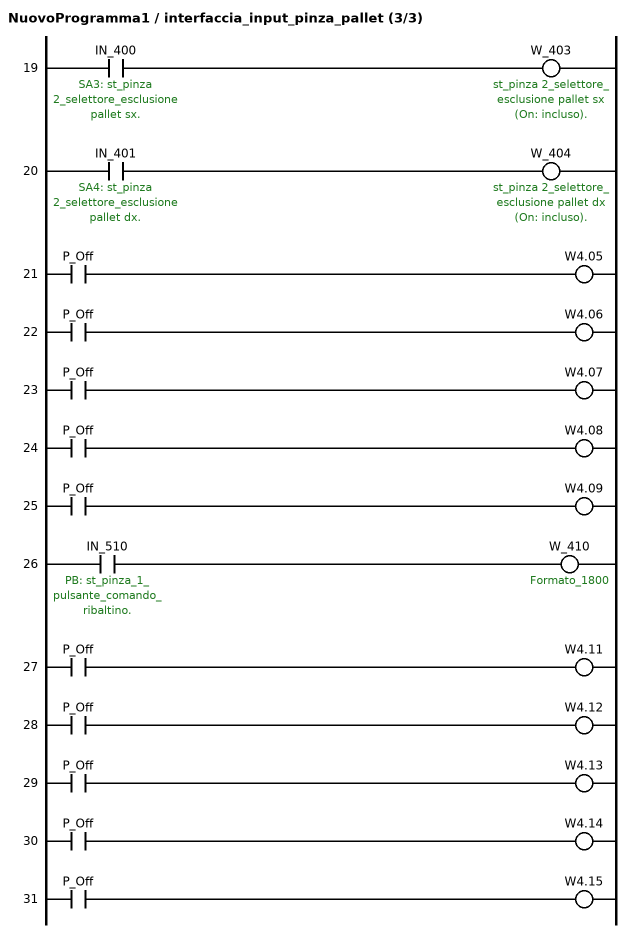
; rung 19
LD IN_400  ; SA3: st_pinza 2_selettore_esclusione pallet sx.
OUT W_403  ; st_pinza 2_selettore_esclusione pallet sx (On: incluso).
; rung 20
LD IN_401  ; SA4: st_pinza 2_selettore_esclusione pallet dx.
OUT W_404  ; st_pinza 2_selettore_esclusione pallet dx (On: incluso).
; rung 21
LD P_Off
OUT W4.05
; rung 22
LD P_Off
OUT W4.06
; rung 23
LD P_Off
OUT W4.07
; rung 24
LD P_Off
OUT W4.08
; rung 25
LD P_Off
OUT W4.09
; rung 26
LD IN_510  ; PB: st_pinza_1_pulsante_comando_ribaltino.
OUT W_410  ; Formato_1800
; rung 27
LD P_Off
OUT W4.11
; rung 28
LD P_Off
OUT W4.12
; rung 29
LD P_Off
OUT W4.13
; rung 30
LD P_Off
OUT W4.14
; rung 31
LD P_Off
OUT W4.15

### Section interfaccia_output

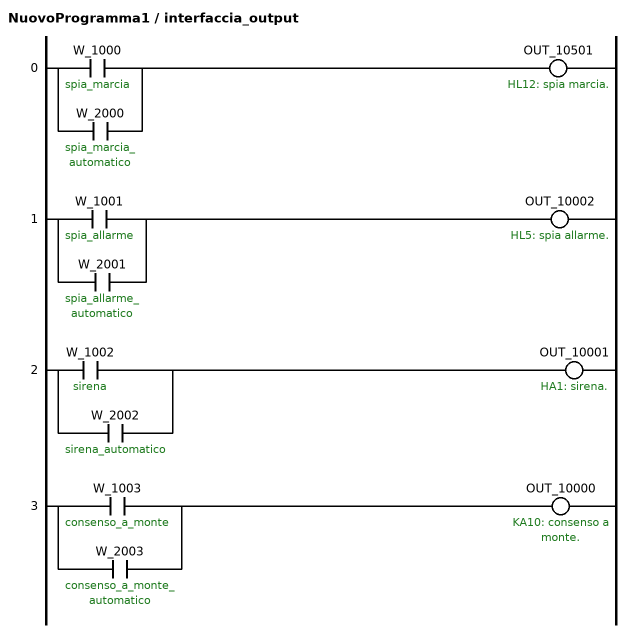
; rung 0
LD W_1000  ; spia_marcia
OR W_2000  ; spia_marcia_automatico
OUT OUT_10501  ; HL12: spia marcia.
; rung 1
LD W_1001  ; spia_allarme
OR W_2001  ; spia_allarme_automatico
OUT OUT_10002  ; HL5: spia allarme.
; rung 2
LD W_1002  ; sirena
OR W_2002  ; sirena_automatico
OUT OUT_10001  ; HA1: sirena.
; rung 3
LD W_1003  ; consenso_a_monte
OR W_2003  ; consenso_a_monte_automatico
OUT OUT_10000  ; KA10: consenso a monte.

### Section interfaccia_output_pinza_ribaltino

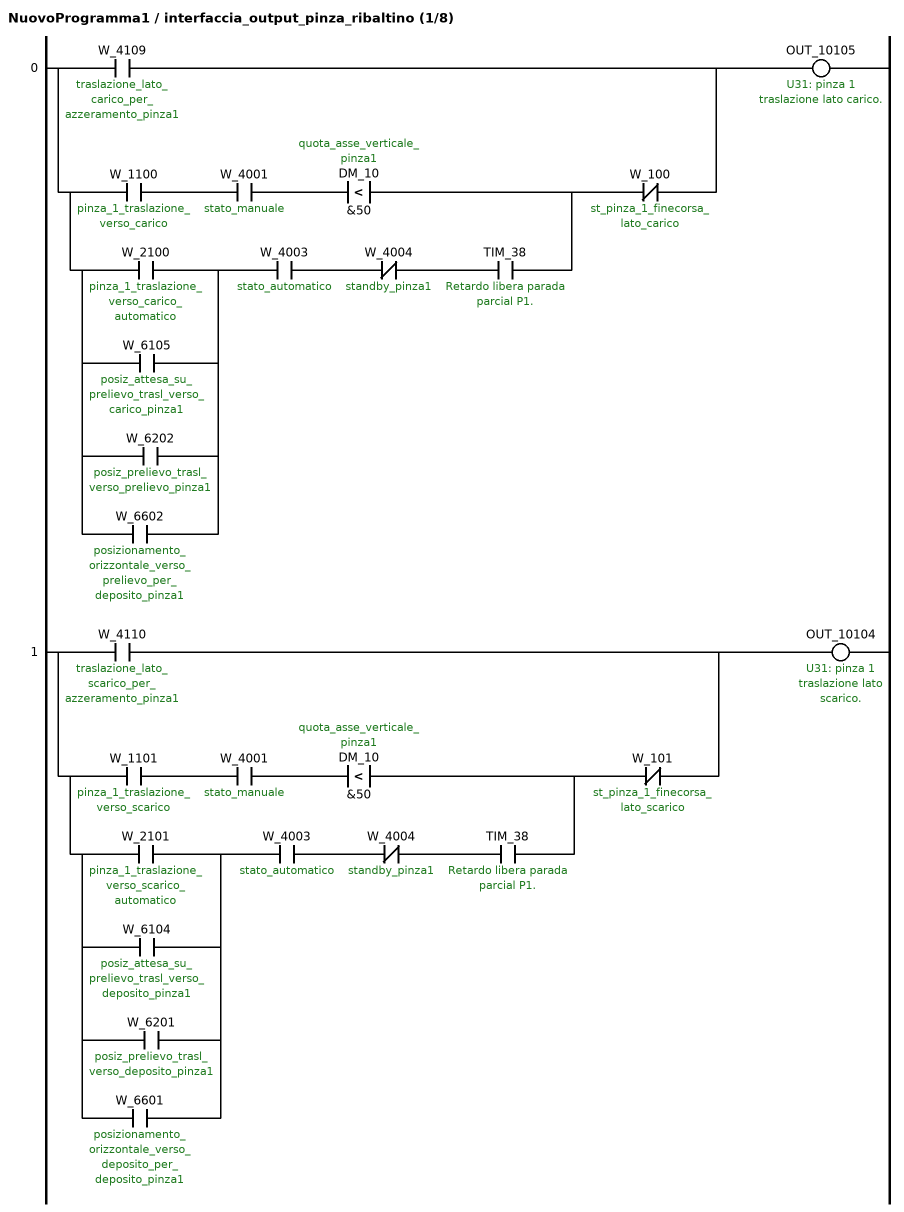
; rung 0
LD W_4109  ; traslazione_lato_carico_per_azzeramento_pinza1
LD W_1100  ; pinza_1_traslazione_verso_carico
AND W_4001  ; stato_manuale
AND<(310) DM_10 &50  ; quota_asse_verticale_pinza1
LD W_2100  ; pinza_1_traslazione_verso_carico_automatico
OR W_6105  ; posiz_attesa_su_prelievo_trasl_verso_carico_pinza1
OR W_6202  ; posiz_prelievo_trasl_verso_prelievo_pinza1
OR W_6602  ; posizionamento_orizzontale_verso_prelievo_per_deposito_pinza1
AND W_4003  ; stato_automatico
ANDNOT W_4004  ; standby_pinza1
AND TIM_38  ; Retardo libera parada parcial P1.
ORLD
ANDNOT W_100  ; st_pinza_1_finecorsa_lato_carico
ORLD
OUT OUT_10105  ; U31: pinza 1 traslazione lato carico.
; rung 1
LD W_4110  ; traslazione_lato_scarico_per_azzeramento_pinza1
LD W_1101  ; pinza_1_traslazione_verso_scarico
AND W_4001  ; stato_manuale
AND<(310) DM_10 &50  ; quota_asse_verticale_pinza1
LD W_2101  ; pinza_1_traslazione_verso_scarico_automatico
OR W_6104  ; posiz_attesa_su_prelievo_trasl_verso_deposito_pinza1
OR W_6201  ; posiz_prelievo_trasl_verso_deposito_pinza1
OR W_6601  ; posizionamento_orizzontale_verso_deposito_per_deposito_pinza1
AND W_4003  ; stato_automatico
ANDNOT W_4004  ; standby_pinza1
AND TIM_38  ; Retardo libera parada parcial P1.
ORLD
ANDNOT W_101  ; st_pinza_1_finecorsa_lato_scarico
ORLD
OUT OUT_10104  ; U31: pinza 1 traslazione lato scarico.

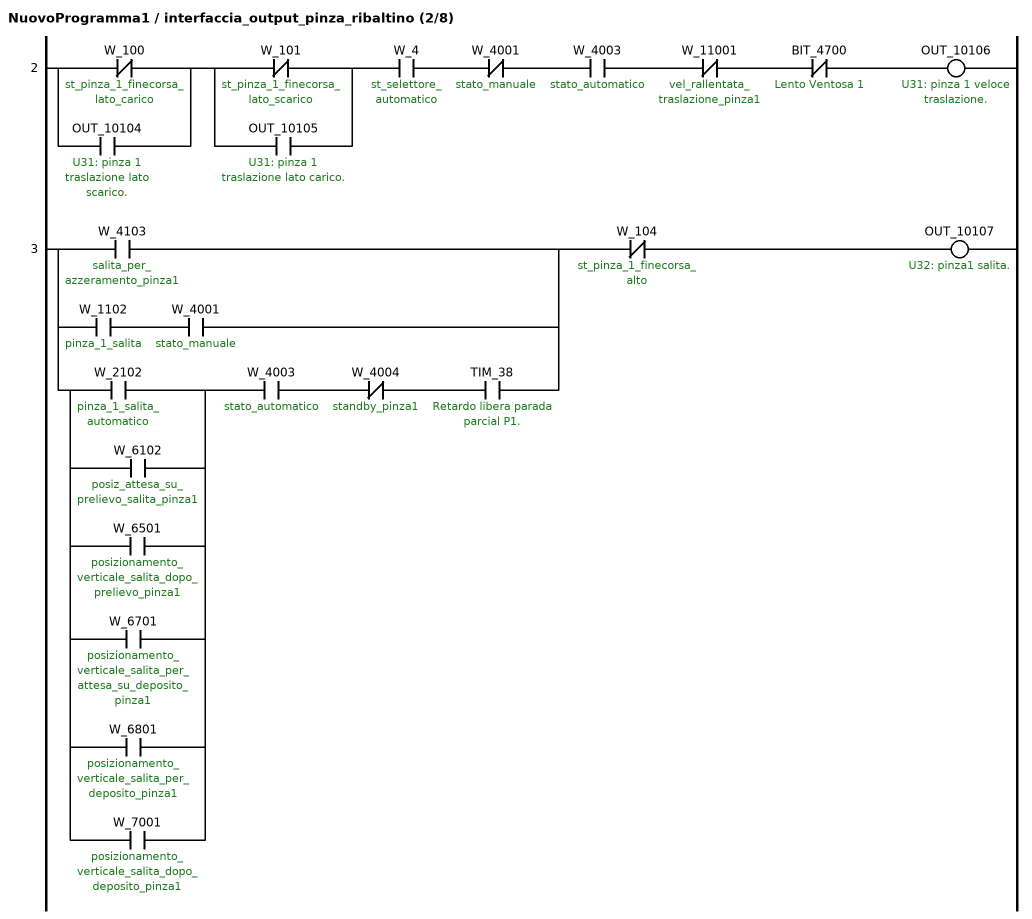
; rung 2
LDNOT W_100  ; st_pinza_1_finecorsa_lato_carico
OR OUT_10104  ; U31: pinza 1 traslazione lato scarico.
LDNOT W_101  ; st_pinza_1_finecorsa_lato_scarico
OR OUT_10105  ; U31: pinza 1 traslazione lato carico.
ANDLD
AND W_4  ; st_selettore_automatico
ANDNOT W_4001  ; stato_manuale
AND W_4003  ; stato_automatico
ANDNOT W_11001  ; vel_rallentata_traslazione_pinza1
ANDNOT BIT_4700  ; Lento Ventosa 1
OUT OUT_10106  ; U31: pinza 1 veloce traslazione.
; rung 3
LD W_4103  ; salita_per_azzeramento_pinza1
LD W_1102  ; pinza_1_salita
AND W_4001  ; stato_manuale
ORLD
LD W_2102  ; pinza_1_salita_automatico
OR W_6102  ; posiz_attesa_su_prelievo_salita_pinza1
OR W_6501  ; posizionamento_verticale_salita_dopo_prelievo_pinza1
OR W_6701  ; posizionamento_verticale_salita_per_attesa_su_deposito_pinza1
OR W_6801  ; posizionamento_verticale_salita_per_deposito_pinza1
OR W_7001  ; posizionamento_verticale_salita_dopo_deposito_pinza1
AND W_4003  ; stato_automatico
ANDNOT W_4004  ; standby_pinza1
AND TIM_38  ; Retardo libera parada parcial P1.
ORLD
ANDNOT W_104  ; st_pinza_1_finecorsa_alto
OUT OUT_10107  ; U32: pinza1 salita.

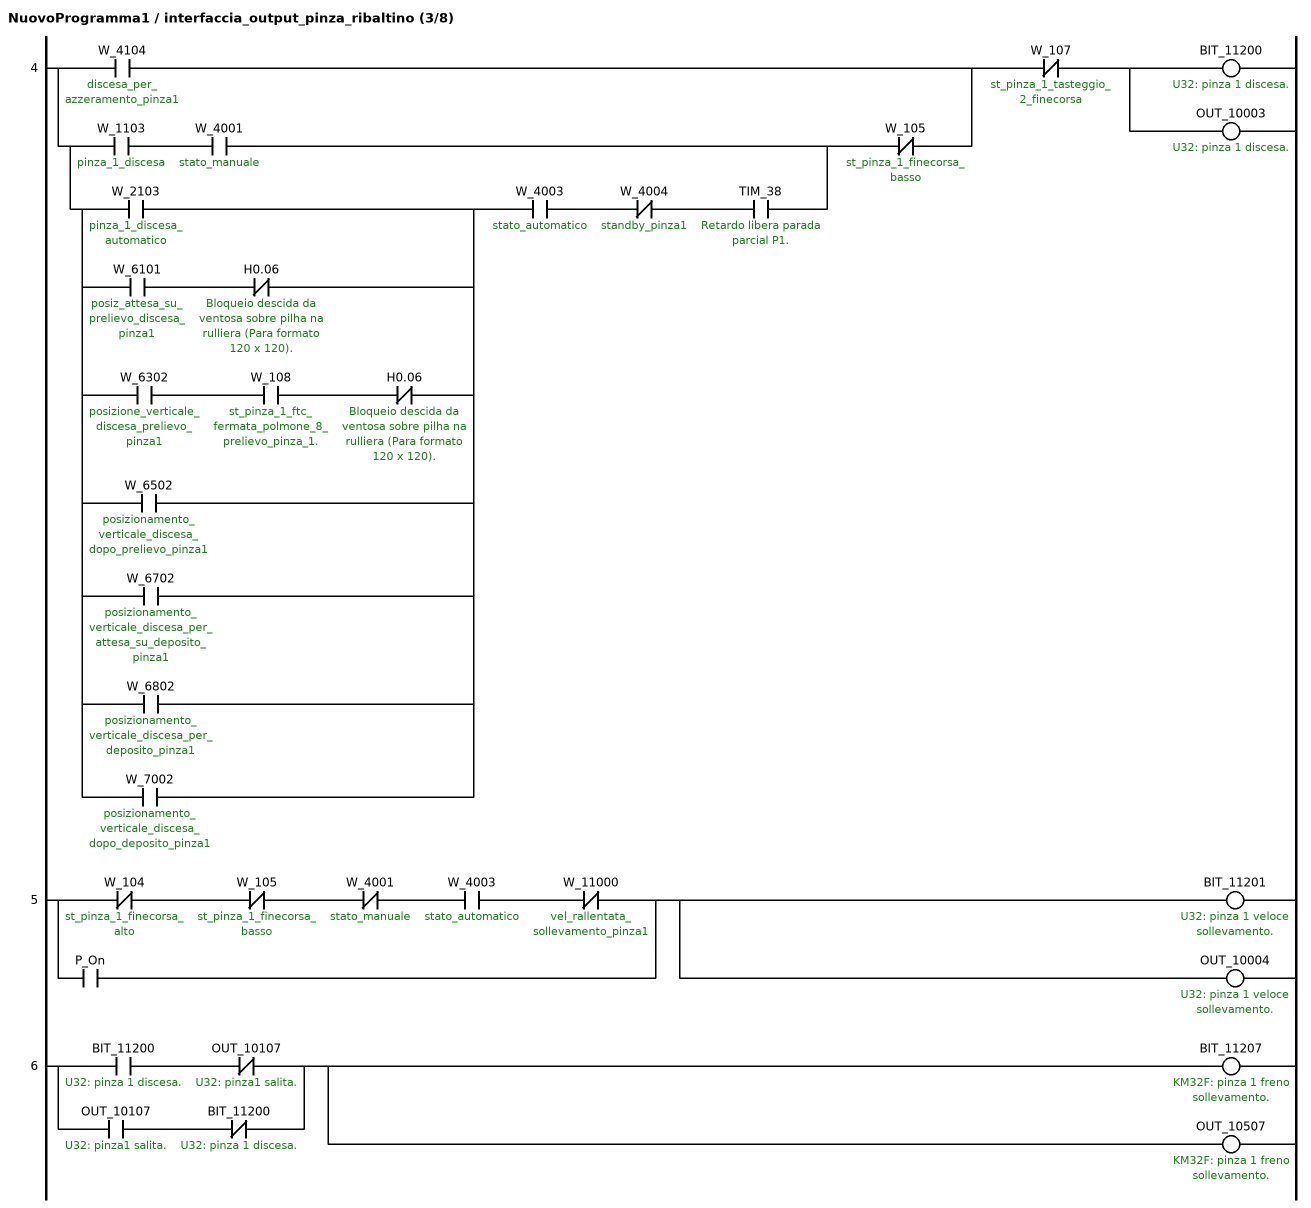
; rung 4
LD W_4104  ; discesa_per_azzeramento_pinza1
LD W_1103  ; pinza_1_discesa
AND W_4001  ; stato_manuale
LD W_2103  ; pinza_1_discesa_automatico
LD W_6101  ; posiz_attesa_su_prelievo_discesa_pinza1
ANDNOT H0.06  ; Bloqueio descida da ventosa sobre pilha na rulliera (Para formato 120 x 120).
ORLD
LD W_6302  ; posizione_verticale_discesa_prelievo_pinza1
AND W_108  ; st_pinza_1_ftc_fermata_polmone_8_prelievo_pinza_1.
ANDNOT H0.06  ; Bloqueio descida da ventosa sobre pilha na rulliera (Para formato 120 x 120).
ORLD
OR W_6502  ; posizionamento_verticale_discesa_dopo_prelievo_pinza1
OR W_6702  ; posizionamento_verticale_discesa_per_attesa_su_deposito_pinza1
OR W_6802  ; posizionamento_verticale_discesa_per_deposito_pinza1
OR W_7002  ; posizionamento_verticale_discesa_dopo_deposito_pinza1
AND W_4003  ; stato_automatico
ANDNOT W_4004  ; standby_pinza1
AND TIM_38  ; Retardo libera parada parcial P1.
ORLD
ANDNOT W_105  ; st_pinza_1_finecorsa_basso
ORLD
ANDNOT W_107  ; st_pinza_1_tasteggio_2_finecorsa
OUT BIT_11200  ; U32: pinza 1 discesa.
OUT OUT_10003  ; U32: pinza 1 discesa.
; rung 5
LDNOT W_104  ; st_pinza_1_finecorsa_alto
ANDNOT W_105  ; st_pinza_1_finecorsa_basso
ANDNOT W_4001  ; stato_manuale
AND W_4003  ; stato_automatico
ANDNOT W_11000  ; vel_rallentata_sollevamento_pinza1
OR P_On
OUT BIT_11201  ; U32: pinza 1 veloce sollevamento.
OUT OUT_10004  ; U32: pinza 1 veloce sollevamento.
; rung 6
LD BIT_11200  ; U32: pinza 1 discesa.
ANDNOT OUT_10107  ; U32: pinza1 salita.
LD OUT_10107  ; U32: pinza1 salita.
ANDNOT BIT_11200  ; U32: pinza 1 discesa.
ORLD
OUT BIT_11207  ; KM32F: pinza 1 freno sollevamento.
OUT OUT_10507  ; KM32F: pinza 1 freno sollevamento.

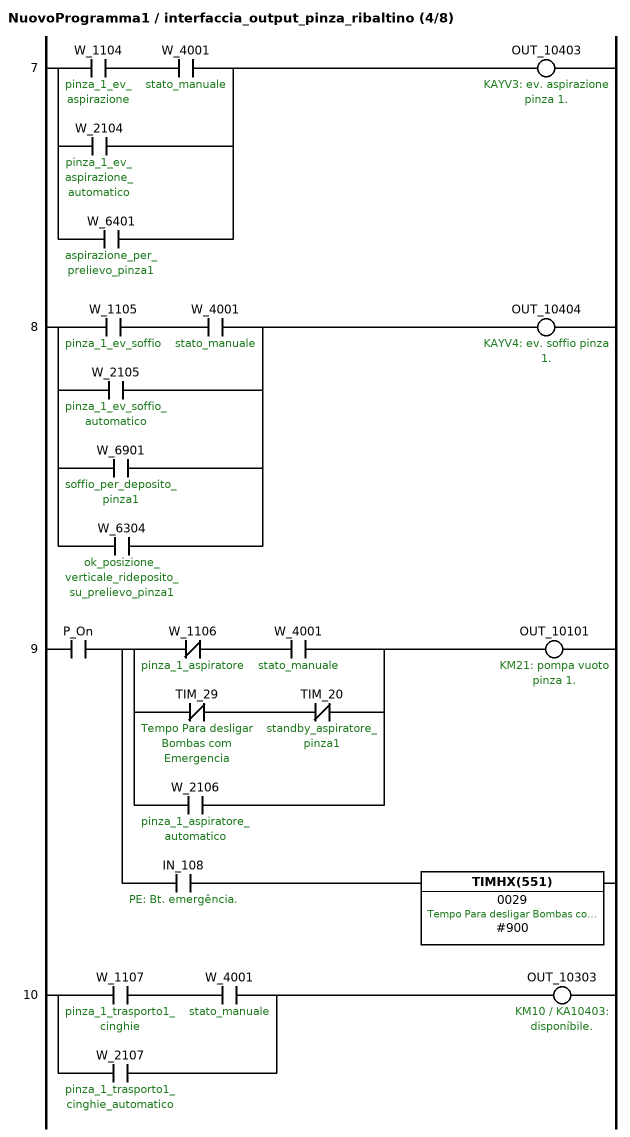
; rung 7
LD W_1104  ; pinza_1_ev_aspirazione
AND W_4001  ; stato_manuale
OR W_2104  ; pinza_1_ev_aspirazione_automatico
OR W_6401  ; aspirazione_per_prelievo_pinza1
OUT OUT_10403  ; KAYV3: ev. aspirazione pinza 1.
; rung 8
LD W_1105  ; pinza_1_ev_soffio
AND W_4001  ; stato_manuale
OR W_2105  ; pinza_1_ev_soffio_automatico
OR W_6901  ; soffio_per_deposito_pinza1
OR W_6304  ; ok_posizione_verticale_rideposito_su_prelievo_pinza1
OUT OUT_10404  ; KAYV4: ev. soffio pinza 1.
; rung 9
LD P_On
OUT TR0
LDNOT W_1106  ; pinza_1_aspiratore
AND W_4001  ; stato_manuale
LDNOT TIM_29  ; Tempo Para desligar Bombas com Emergencia
ANDNOT TIM_20  ; standby_aspiratore_pinza1
ORLD
OR W_2106  ; pinza_1_aspiratore_automatico
ANDLD
OUT OUT_10101  ; KM21: pompa vuoto pinza 1.
LD TR0
AND IN_108  ; PE: Bt. emergência.
TIMHX(551) 0029 #900  ; Tempo Para desligar Bombas com Emergencia
; rung 10
LD W_1107  ; pinza_1_trasporto1_cinghie
AND W_4001  ; stato_manuale
OR W_2107  ; pinza_1_trasporto1_cinghie_automatico
OUT OUT_10303  ; KM10 / KA10403: disponíbile.

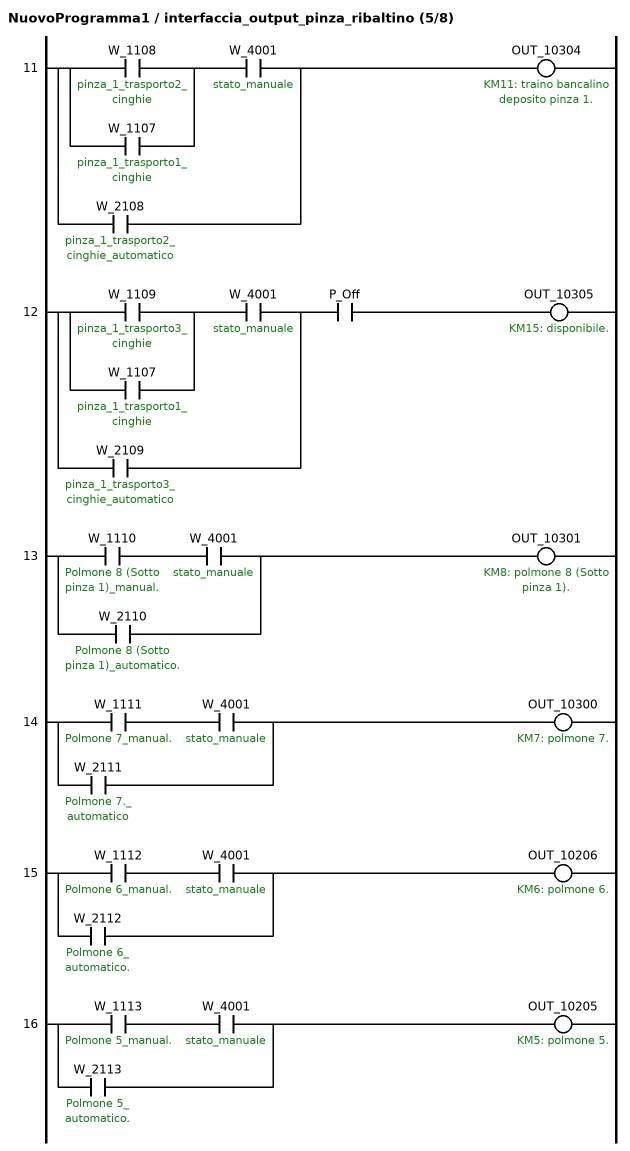
; rung 11
LD W_1108  ; pinza_1_trasporto2_cinghie
OR W_1107  ; pinza_1_trasporto1_cinghie
AND W_4001  ; stato_manuale
OR W_2108  ; pinza_1_trasporto2_cinghie_automatico
OUT OUT_10304  ; KM11: traino bancalino deposito pinza 1.
; rung 12
LD W_1109  ; pinza_1_trasporto3_cinghie
OR W_1107  ; pinza_1_trasporto1_cinghie
AND W_4001  ; stato_manuale
OR W_2109  ; pinza_1_trasporto3_cinghie_automatico
AND P_Off
OUT OUT_10305  ; KM15: disponibile.
; rung 13
LD W_1110  ; Polmone 8 (Sotto pinza 1)_manual.
AND W_4001  ; stato_manuale
OR W_2110  ; Polmone 8 (Sotto pinza 1)_automatico.
OUT OUT_10301  ; KM8: polmone 8 (Sotto pinza 1).
; rung 14
LD W_1111  ; Polmone 7_manual.
AND W_4001  ; stato_manuale
OR W_2111  ; Polmone 7._automatico
OUT OUT_10300  ; KM7: polmone 7.
; rung 15
LD W_1112  ; Polmone 6_manual.
AND W_4001  ; stato_manuale
OR W_2112  ; Polmone 6_automatico.
OUT OUT_10206  ; KM6: polmone 6.
; rung 16
LD W_1113  ; Polmone 5_manual.
AND W_4001  ; stato_manuale
OR W_2113  ; Polmone 5_automatico.
OUT OUT_10205  ; KM5: polmone 5.

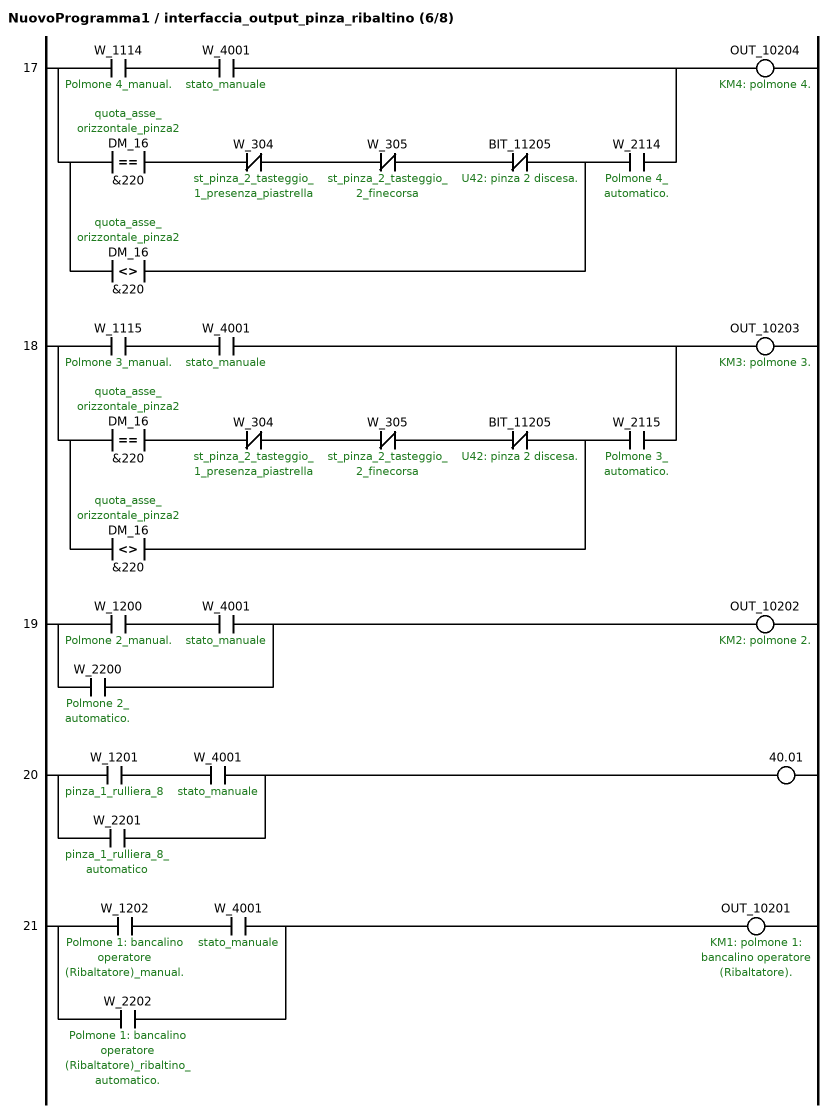
; rung 17
LD W_1114  ; Polmone 4_manual.
AND W_4001  ; stato_manuale
LD=(300) DM_16 &220  ; quota_asse_orizzontale_pinza2
ANDNOT W_304  ; st_pinza_2_tasteggio_1_presenza_piastrella
ANDNOT W_305  ; st_pinza_2_tasteggio_2_finecorsa
ANDNOT BIT_11205  ; U42: pinza 2 discesa.
OR<>(305) DM_16 &220  ; quota_asse_orizzontale_pinza2
AND W_2114  ; Polmone 4_automatico.
ORLD
OUT OUT_10204  ; KM4: polmone 4.
; rung 18
LD W_1115  ; Polmone 3_manual.
AND W_4001  ; stato_manuale
LD=(300) DM_16 &220  ; quota_asse_orizzontale_pinza2
ANDNOT W_304  ; st_pinza_2_tasteggio_1_presenza_piastrella
ANDNOT W_305  ; st_pinza_2_tasteggio_2_finecorsa
ANDNOT BIT_11205  ; U42: pinza 2 discesa.
OR<>(305) DM_16 &220  ; quota_asse_orizzontale_pinza2
AND W_2115  ; Polmone 3_automatico.
ORLD
OUT OUT_10203  ; KM3: polmone 3.
; rung 19
LD W_1200  ; Polmone 2_manual.
AND W_4001  ; stato_manuale
OR W_2200  ; Polmone 2_automatico.
OUT OUT_10202  ; KM2: polmone 2.
; rung 20
LD W_1201  ; pinza_1_rulliera_8
AND W_4001  ; stato_manuale
OR W_2201  ; pinza_1_rulliera_8_automatico
OUT 40.01
; rung 21
LD W_1202  ; Polmone 1: bancalino operatore (Ribaltatore)_manual.
AND W_4001  ; stato_manuale
OR W_2202  ; Polmone 1: bancalino operatore (Ribaltatore)_ribaltino_automatico.
OUT OUT_10201  ; KM1: polmone 1: bancalino operatore (Ribaltatore).

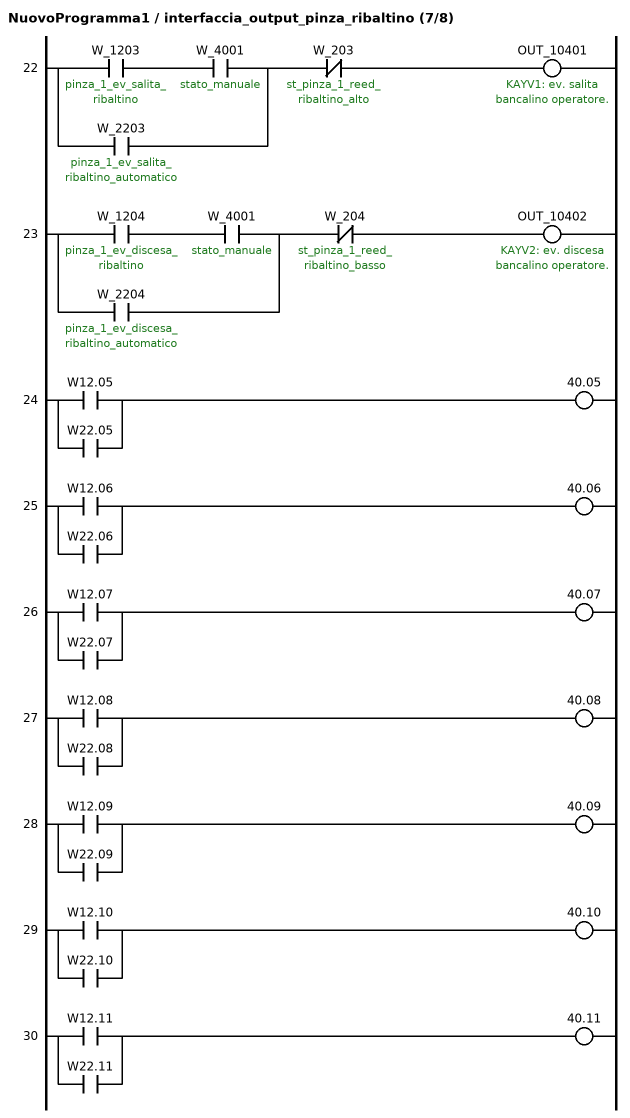
; rung 22
LD W_1203  ; pinza_1_ev_salita_ribaltino
AND W_4001  ; stato_manuale
OR W_2203  ; pinza_1_ev_salita_ribaltino_automatico
ANDNOT W_203  ; st_pinza_1_reed_ribaltino_alto
OUT OUT_10401  ; KAYV1: ev. salita bancalino operatore.
; rung 23
LD W_1204  ; pinza_1_ev_discesa_ribaltino
AND W_4001  ; stato_manuale
OR W_2204  ; pinza_1_ev_discesa_ribaltino_automatico
ANDNOT W_204  ; st_pinza_1_reed_ribaltino_basso
OUT OUT_10402  ; KAYV2: ev. discesa bancalino operatore.
; rung 24
LD W12.05
OR W22.05
OUT 40.05
; rung 25
LD W12.06
OR W22.06
OUT 40.06
; rung 26
LD W12.07
OR W22.07
OUT 40.07
; rung 27
LD W12.08
OR W22.08
OUT 40.08
; rung 28
LD W12.09
OR W22.09
OUT 40.09
; rung 29
LD W12.10
OR W22.10
OUT 40.10
; rung 30
LD W12.11
OR W22.11
OUT 40.11

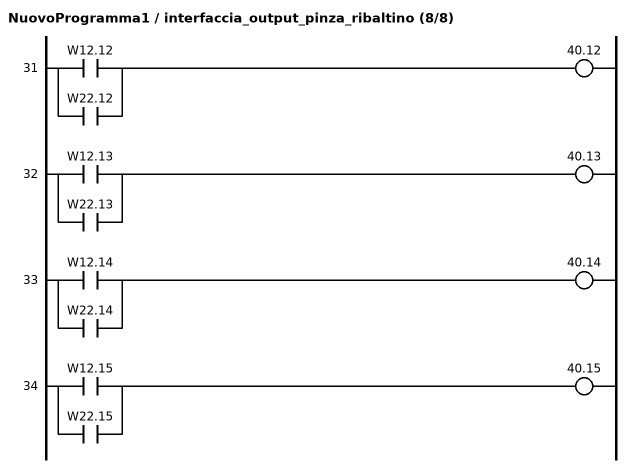
; rung 31
LD W12.12
OR W22.12
OUT 40.12
; rung 32
LD W12.13
OR W22.13
OUT 40.13
; rung 33
LD W12.14
OR W22.14
OUT 40.14
; rung 34
LD W12.15
OR W22.15
OUT 40.15

### Section interfaccia_output_pinza_pallet

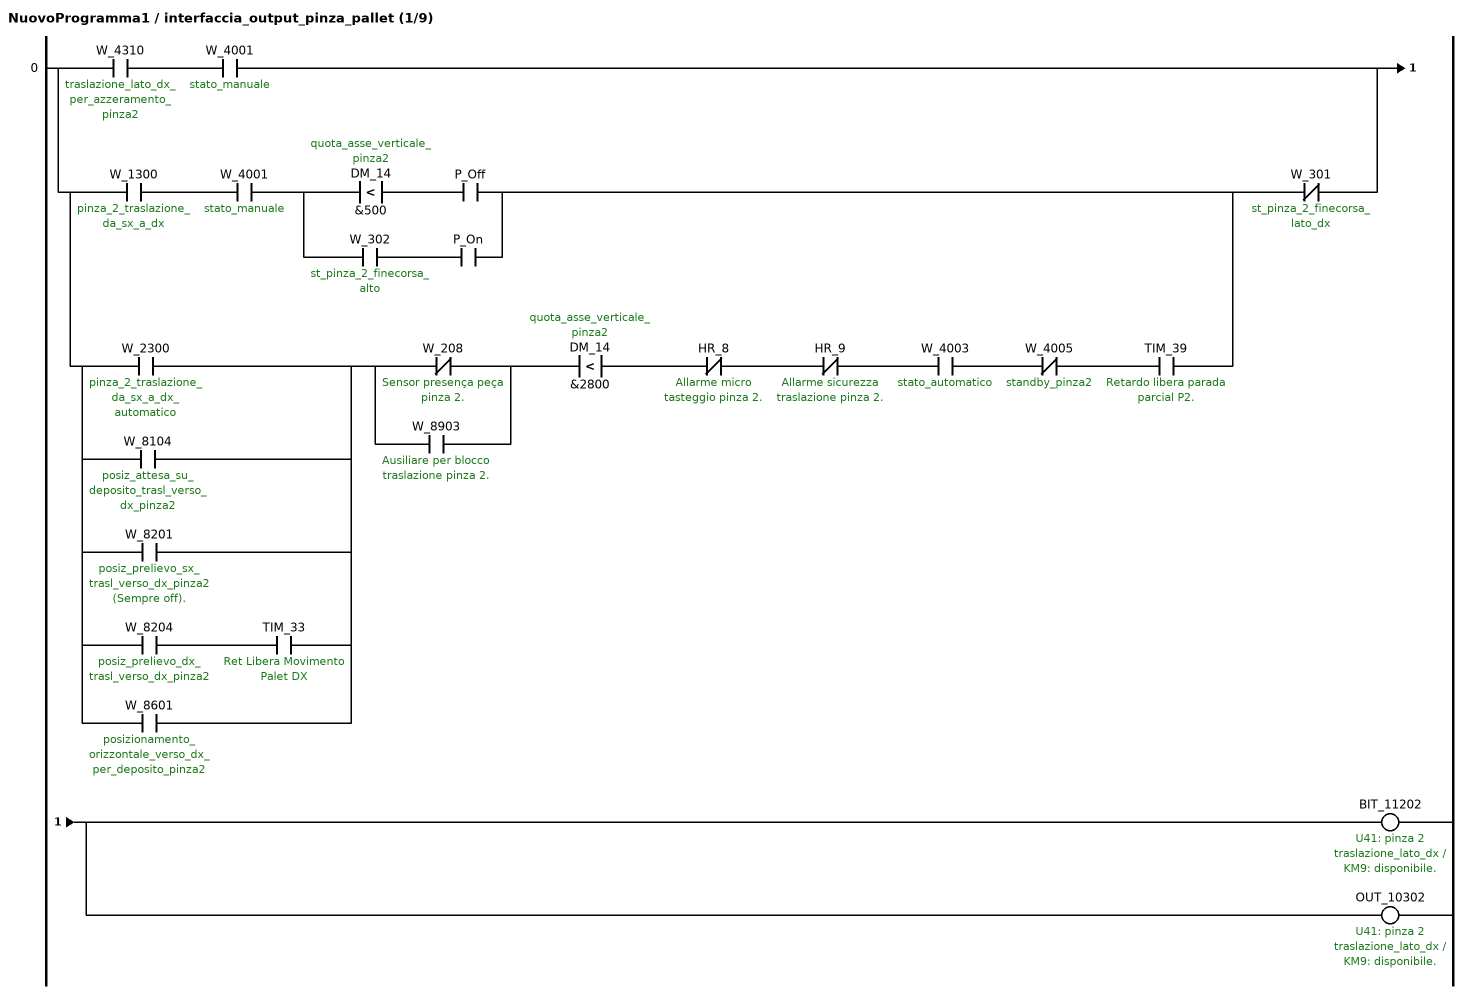
; rung 0
LD W_4310  ; traslazione_lato_dx_per_azzeramento_pinza2
AND W_4001  ; stato_manuale
LD W_1300  ; pinza_2_traslazione_da_sx_a_dx
AND W_4001  ; stato_manuale
LD<(310) DM_14 &500  ; quota_asse_verticale_pinza2
AND P_Off
LD W_302  ; st_pinza_2_finecorsa_alto
AND P_On
ORLD
ANDLD
LD W_2300  ; pinza_2_traslazione_da_sx_a_dx_automatico
OR W_8104  ; posiz_attesa_su_deposito_trasl_verso_dx_pinza2
OR W_8201  ; posiz_prelievo_sx_trasl_verso_dx_pinza2 (Sempre off).
LD W_8204  ; posiz_prelievo_dx_trasl_verso_dx_pinza2
AND TIM_33  ; Ret Libera Movimento Palet DX
ORLD
OR W_8601  ; posizionamento_orizzontale_verso_dx_per_deposito_pinza2
LDNOT W_208  ; Sensor presença peça pinza 2.
OR W_8903  ; Ausiliare per blocco traslazione pinza 2.
ANDLD
AND<S(312) DM_14 &2800  ; quota_asse_verticale_pinza2
ANDNOT HR_8  ; Allarme micro tasteggio pinza 2.
ANDNOT HR_9  ; Allarme sicurezza traslazione pinza 2.
AND W_4003  ; stato_automatico
ANDNOT W_4005  ; standby_pinza2
AND TIM_39  ; Retardo libera parada parcial P2.
ORLD
ANDNOT W_301  ; st_pinza_2_finecorsa_lato_dx
ORLD
OUT BIT_11202  ; U41: pinza 2 traslazione_lato_dx / KM9: disponibile.
OUT OUT_10302  ; U41: pinza 2 traslazione_lato_dx / KM9: disponibile.

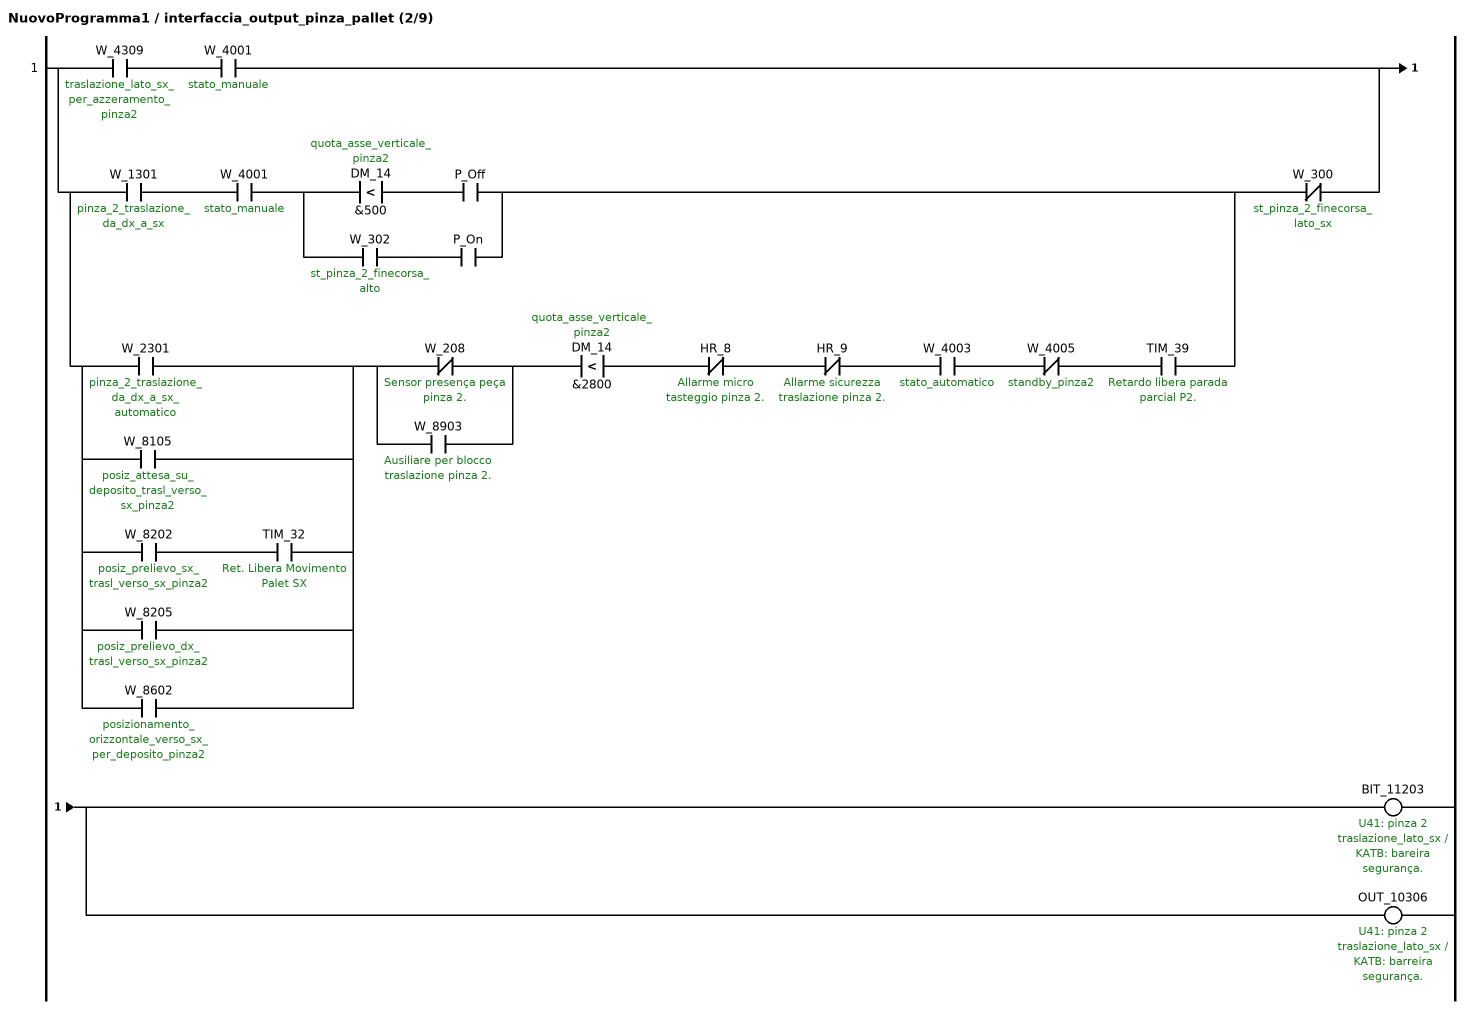
; rung 1
LD W_4309  ; traslazione_lato_sx_per_azzeramento_pinza2
AND W_4001  ; stato_manuale
LD W_1301  ; pinza_2_traslazione_da_dx_a_sx
AND W_4001  ; stato_manuale
LD<(310) DM_14 &500  ; quota_asse_verticale_pinza2
AND P_Off
LD W_302  ; st_pinza_2_finecorsa_alto
AND P_On
ORLD
ANDLD
LD W_2301  ; pinza_2_traslazione_da_dx_a_sx_automatico
OR W_8105  ; posiz_attesa_su_deposito_trasl_verso_sx_pinza2
LD W_8202  ; posiz_prelievo_sx_trasl_verso_sx_pinza2
AND TIM_32  ; Ret. Libera Movimento Palet SX
ORLD
OR W_8205  ; posiz_prelievo_dx_trasl_verso_sx_pinza2
OR W_8602  ; posizionamento_orizzontale_verso_sx_per_deposito_pinza2
LDNOT W_208  ; Sensor presença peça pinza 2.
OR W_8903  ; Ausiliare per blocco traslazione pinza 2.
ANDLD
AND<S(312) DM_14 &2800  ; quota_asse_verticale_pinza2
ANDNOT HR_8  ; Allarme micro tasteggio pinza 2.
ANDNOT HR_9  ; Allarme sicurezza traslazione pinza 2.
AND W_4003  ; stato_automatico
ANDNOT W_4005  ; standby_pinza2
AND TIM_39  ; Retardo libera parada parcial P2.
ORLD
ANDNOT W_300  ; st_pinza_2_finecorsa_lato_sx
ORLD
OUT BIT_11203  ; U41: pinza 2 traslazione_lato_sx / KATB: bareira segurança.
OUT OUT_10306  ; U41: pinza 2 traslazione_lato_sx / KATB: barreira segurança.

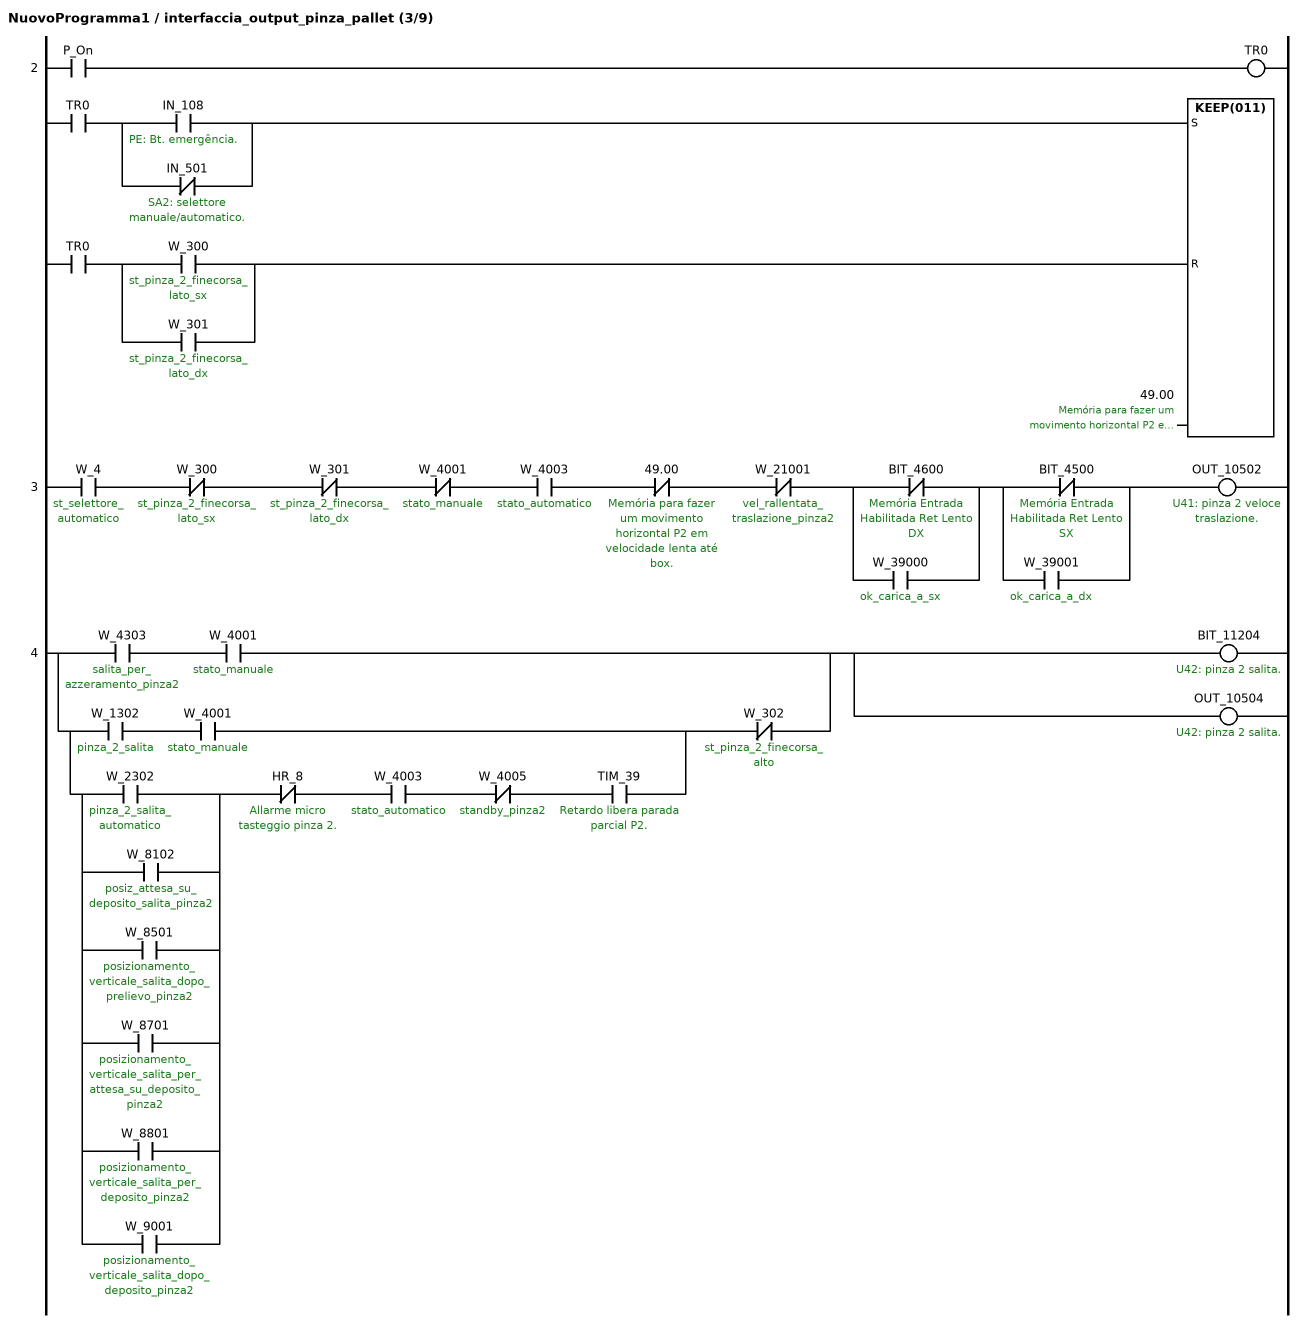
; rung 2
LD P_On
OUT TR0
LD IN_108  ; PE: Bt. emergência.
ORNOT IN_501  ; SA2: selettore manuale/automatico.
ANDLD
LD TR0
LD W_300  ; st_pinza_2_finecorsa_lato_sx
OR W_301  ; st_pinza_2_finecorsa_lato_dx
ANDLD
KEEP(011) 49.00  ; Memória para fazer um movimento horizontal P2 em velocidade lenta até box.
; rung 3
LD W_4  ; st_selettore_automatico
ANDNOT W_300  ; st_pinza_2_finecorsa_lato_sx
ANDNOT W_301  ; st_pinza_2_finecorsa_lato_dx
ANDNOT W_4001  ; stato_manuale
AND W_4003  ; stato_automatico
ANDNOT 49.00  ; Memória para fazer um movimento horizontal P2 em velocidade lenta até box.
ANDNOT W_21001  ; vel_rallentata_traslazione_pinza2
LDNOT BIT_4600  ; Memória Entrada Habilitada Ret Lento DX
OR W_39000  ; ok_carica_a_sx
ANDLD
LDNOT BIT_4500  ; Memória Entrada Habilitada Ret Lento SX
OR W_39001  ; ok_carica_a_dx
ANDLD
OUT OUT_10502  ; U41: pinza 2 veloce traslazione.
; rung 4
LD W_4303  ; salita_per_azzeramento_pinza2
AND W_4001  ; stato_manuale
LD W_1302  ; pinza_2_salita
AND W_4001  ; stato_manuale
LD W_2302  ; pinza_2_salita_automatico
OR W_8102  ; posiz_attesa_su_deposito_salita_pinza2
OR W_8501  ; posizionamento_verticale_salita_dopo_prelievo_pinza2
OR W_8701  ; posizionamento_verticale_salita_per_attesa_su_deposito_pinza2
OR W_8801  ; posizionamento_verticale_salita_per_deposito_pinza2
OR W_9001  ; posizionamento_verticale_salita_dopo_deposito_pinza2
ANDNOT HR_8  ; Allarme micro tasteggio pinza 2.
AND W_4003  ; stato_automatico
ANDNOT W_4005  ; standby_pinza2
AND TIM_39  ; Retardo libera parada parcial P2.
ORLD
ANDNOT W_302  ; st_pinza_2_finecorsa_alto
ORLD
OUT BIT_11204  ; U42: pinza 2 salita.
OUT OUT_10504  ; U42: pinza 2 salita.

